IF NOT bRun THEN
	iSecondDoseCount				:= 0;
	bCycleDone 					:= FALSE;
	bCycleNotDone 				:= FALSE;	
END_IF
	
// ZASYWANIE PRZY ZJEZDZIE W DÓŁ
IF NOT bSucking AND bDoSmallSucking THEN
	mcDispencerMoveAbsolute1.Execute:= bDosingValveClosedSensor; 
	mcDispencerMoveAbsolute1.Velocity:= lrSuckVelocity;
	mcDispencerMoveAbsolute1.Position:= lrDoseVolume + 3;
	mcDispencerMoveAbsolute1.Acceleration:= lrSuckAcceleration;
	mcDispencerMoveAbsolute1.Deceleration:= lrSuckDeceleration;
	IF mcDispencerMoveAbsolute1.Done THEN
		bDoSmallSucking						:=	FALSE;
		bDoSmallSuckingDone					:=	TRUE;	
		mcDispencerMoveAbsolute1.Execute	:=	FALSE;
	END_IF
END_IF
IF  bSucking AND tonSuckValveCloseTimeDelay.Q  THEN  // [4] Opóżnienie zamknięcia zaworu ssącego [ms]                            
		bSucking := FALSE;
		mcDispencerMoveAbsolute1.Execute:= FALSE;
		bSuckingValveActuator:=FALSE;
END_IF	

ManualMovementsCleaning();
ManualMovementsPulling();
ManualMovementSync();

//ZABEZPIECZENIE PRZED UDERZENIEM W TACKĘ OCIEKOWĄ
IF DispencerLifterAxisRef.NcToPlc.ActPos	<	(lrDropCatcherHeightCV+lrDropCatcherOpenDistance-5) AND NOT bDropCatcherBackSensor THEN
	mcLifterManualMove.JogBackwards:=FALSE;
END_IF

IF (DispencerLifterAxisRef.NcToPlc.ActPos  <= 	lrDropCatcherHeightCV+(lrDropCatcherOpenDistance-5))  THEN 
	bDropCatcherActuator:=FALSE;
END_IF
END_ACTION

ACTION ManualMovementsCleaning:

(*****************CYKL MYCIA DOZOWNIKA*******************
eCleaningPreparing:=18,	//Mycie | przejazd do pozycji górnej
eCleaningReady:=19,		//Mycie | pozycja tłoka w górze
eCleaning:=20,			//Mycie | w trakcie ruchu w dół
eCleaningDone:=21		//Mycie | pozycja tłoka w dole
*********************************************************)

// Włączenie mycia
IF bManualCleaningMode  AND  (	NOT (eRunningState	=	E_DispencerState.eCleaningPreparing)		AND
								NOT (eRunningState	=	E_DispencerState.eCleaningReady) 			AND
								NOT (eRunningState	=	E_DispencerState.eCleaning)					AND
								NOT (eRunningState	=	E_DispencerState.eCleaningDone) )			THEN 
	eRunningState	:=	E_DispencerState.eCleaningPreparing;	
END_IF

//Wyłączenie mycia, zatrzymywanie
IF NOT bManualCleaningMode AND  (	eRunningState	=	E_DispencerState.eCleaningReady OR
									eRunningState	=	E_DispencerState.eCleaning OR
									eRunningState	=	E_DispencerState.eCleaningDone )	THEN

	mcDispencerStop.Execute					:= TRUE;
	bSuckingValveActuator					:= FALSE;	
	bDosingValveActuator					:= FALSE;	
	IF 	mcDispencerStop.Done THEN			
		mcDispencerStop.Execute				:= FALSE;
		eState								:= E_Station.eManualMovement;
		eRunningState						:= E_DispencerState.eReady;
	END_IF	
END_IF


//Przygotowanie
IF eRunningState=E_DispencerState.eCleaningPreparing THEN
	bSuckingValveActuator					:= TRUE;
	bDosingValveActuator					:= FALSE;
	mcDispencerMoveAbsolute1.Velocity		:= (lrDosePhase2Velocity*2)		*1.8; 	//Prędkość brana z receptury zwiększona o 30% i 2x większa niż dozowania
	mcDispencerMoveAbsolute1.Acceleration	:= lrDosePhase2Acceleration		*1.8;
	mcDispencerMoveAbsolute1.Deceleration	:= lrDosePhase2Acceleration		*1.8;
	mcDispencerMoveAbsolute1.Position		:= lrRatedDose;
	mcDispencerMoveAbsolute1.Execute		:= bSuckingValveActuator AND bSuckingValveOpenedSensor AND bDosingValveClosedSensor ;
	IF mcDispencerMoveAbsolute1.Done THEN
		mcDispencerMoveAbsolute1.Execute	:= FALSE;
		eRunningState								:= E_DispencerState.eCleaningReady;
	END_IF
END_IF


//Gotowość do mycia
IF eRunningState=E_DispencerState.eCleaningReady THEN
	bSuckingValveActuator					:= FALSE;
	bDosingValveActuator					:= FALSE;
	IF bManualCleaning THEN
		eRunningState								:= E_DispencerState.eCleaning;
	END_IF
END_IF


//Mycie, ruch w dół
IF eRunningState=E_DispencerState.eCleaning THEN
	bSuckingValveActuator					:= FALSE;
	bDosingValveActuator					:= TRUE;
	mcDispencerMoveAbsolute2.Velocity		:= lrDosePhase2Velocity			*1.8;
	mcDispencerMoveAbsolute2.Acceleration	:= lrDosePhase2Acceleration		*1.8;
	mcDispencerMoveAbsolute2.Deceleration	:= lrDosePhase2Acceleration		*1.8;
	mcDispencerMoveAbsolute2.Position		:= 0;
	mcDispencerMoveAbsolute2.Execute		:= bDosingValveActuator AND bSuckingValveClosedSensor AND bDosingValveOpenedSensor;
	IF mcDispencerMoveAbsolute2.Done THEN
		mcDispencerMoveAbsolute2.Execute	:= FALSE;
		eRunningState								:= E_DispencerState.eCleaningDone;
	END_IF	
END_IF


//Koniec mycia
IF eRunningState=E_DispencerState.eCleaningDone THEN
	bSuckingValveActuator					:= FALSE;
	bDosingValveActuator					:= FALSE;
	IF NOT bManualCleaning THEN
		eRunningState								:= E_DispencerState.eCleaningPreparing;
	END_IF
END_IF
END_ACTION

ACTION ManualMovementsPulling:
//CYKL PRZECIĄGANIA MASY
IF eRunningState=E_DispencerState.ePulling THEN
	
	IF NOT bManualPullingFast AND NOT bManualPullingSlow AND NOT bSuckingValveActuator AND NOT bDosingValveActuator AND bSuckingValveClosedSensor AND bDosingValveClosedSensor AND mcDispencerStop.Done THEN
		mcDispencerStop.Execute:=FALSE;
		mcDispencerMoveAbsolute1.Execute:=FALSE;
		mcDispencerMoveAbsolute2.Execute:=FALSE;
		bSuckingValveActuator:=FALSE;
		bDosingValveActuator:=FALSE;
		bManualPullingLatch:=FALSE;
		mcLifterManualMove.JogForward:=FALSE;
		mcLifterManualMove.JogBackwards:= FALSE;
		eState:=E_Station.eManualMovement;
		eRunningState:=E_DispencerState.eReady;
	END_IF

	mcDispencerMoveAbsolute1.Execute:=bSuckingValveActuator AND bSuckingValveOpenedSensor AND bDosingValveClosedSensor AND (bManualPullingFast OR bManualPullingSlow);
	IF mcDispencerMoveAbsolute1.Execute THEN
		;
	END_IF
	mcDispencerMoveAbsolute2.Execute:=bDosingValveActuator AND bSuckingValveClosedSensor AND bDosingValveOpenedSensor AND (bManualPullingFast OR bManualPullingSlow);
	IF bManualPullingFast THEN
		lrPullingVelocity:=300;
	ELSIF bManualPullingSlow THEN
		lrPullingVelocity:=100;
	END_IF
	mcDispencerMoveAbsolute1.Velocity:=lrPullingVelocity;
	mcDispencerMoveAbsolute2.Velocity:=lrPullingVelocity;
	
	mcDispencerMoveAbsolute1.Acceleration:=800;
	mcDispencerMoveAbsolute2.Acceleration:=800;
	mcDispencerMoveAbsolute1.Deceleration:=800;
	mcDispencerMoveAbsolute2.Deceleration:=800;
	mcDispencerMoveAbsolute1.Position:=lrRatedDose;
	mcDispencerMoveAbsolute2.Position:=0;
	
	bSuckingValveActuator:= NOT mcDispencerMoveAbsolute1.DONE AND NOT bDosingValveActuator AND  (bManualPullingFast OR bManualPullingSlow);
	bDosingValveActuator:= NOT mcDispencerMoveAbsolute2.DONE AND NOT bSuckingValveActuator AND (bManualPullingFast OR bManualPullingSlow OR mcDispencerMoveAbsolute2.Busy);
	mcDispencerStop.Execute:=NOT bSuckingValveActuator AND NOT bDosingValveActuator AND NOT bManualPullingFast AND NOT bManualPullingSlow AND eRunningState=E_DispencerState.ePulling;
END_IF
END_ACTION

ACTION ManualMovementsStepMode:
bManualLifterUp;
bManualLifterDown;
bStepMode;		
lrSetPosStepMode;

// Limity
IF lrSetPosStepMode < 1			THEN	lrSetPosStepMode := 1;	END_IF
IF lrSetPosStepMode > 10		THEN	lrSetPosStepMode := 10;	END_IF

// Zabezpieczenie przed zbyt szybkim włączaniem
tofStepModeMoving				(IN := bStepModeMoving,					PT:=T#500MS);

// Możliwe włączenie jeżeli zakończyło poprzedni ruch
rtStepModeUp					(CLK :=	bStepMode AND NOT tofStepModeMoving.Q	AND bManualLifterUp,	Q=>);
rtStepModeDown					(CLK :=	bStepMode AND NOT tofStepModeMoving.Q 	AND bManualLifterDown,	Q=>);

// Włączenie ruchu w górę
IF rtStepModeUp.Q THEN
	bStepModeMoving				:= TRUE;
	lrStepModeHeightMotorSV		:= lrLifterActualPosition	+	lrSetPosStepMode;
END_IF

// Włączenie ruchu w dół
IF rtStepModeDown.Q THEN
	bStepModeMoving				:= TRUE;
	lrStepModeHeightMotorSV		:= lrLifterActualPosition	-	lrSetPosStepMode;
END_IF
// DODAĆ RESET bStepModeMoving PO BLEDZIE!
// Ruch w górę !SPRAWDZIC ZNAKI!
IF bStepModeMoving THEN
	mcLifterManualMove.JogForward		:=	lrLifterActualPosition	<=	lrStepModeHeightMotorSV;
	mcLifterManualMove.JogBackwards		:=	lrLifterActualPosition	>=	lrStepModeHeightMotorSV;	
	
	IF ABS(lrLifterActualPosition-lrStepModeHeightMotorSV) < 0.5	OR	// Pozycja osiągnięta (co do 1mm)
			(lrLifterActualPosition<=lrMinPosition)					OR 	// Pozycja poniżej minimalnej
			(lrLifterActualPosition>=lrMaxPosition) 					// Pozycja powyżej maksymalnej
	THEN
		mcLifterManualMove.JogForward	:= FALSE;
		mcLifterManualMove.JogForward	:= FALSE;
		bStepModeMoving					:= FALSE;
		bManualLifterUp					:= FALSE;
		bManualLifterDown				:= FALSE;
	END_IF	
END_IF
END_ACTION

ACTION ManualMovementSync:
//Przygotowanie
IF bManualSync THEN
	
CASE iManualSyncCase OF
	
	0:	
		//Rozpoczęcie
		IF bManualSync THEN
			iManualSyncCase	:=	iManualSyncCase	+	10;
		END_IF

	10:
		
			//Ruch tłokiem
			IF ABS(DispencerAxisRef.NcToPlc.ActPos-lrDoseVolume)>1 THEN //Nie wykonuj nie potrzebnie ruchu jeżeli już jest na pozycji
				bSuckingValveActuator				:= ABS(DispencerAxisRef.NcToPlc.ActPos-lrDoseVolume)>1;
			END_IF
			bDosingValveActuator					:= FALSE;
			mcDispencerMoveAbsolute1.Velocity		:= (lrDosePhase2Velocity*2)		*1.8; 	//Prędkość brana z receptury zwiększona o 30% i 2x większa niż dozowania
			mcDispencerMoveAbsolute1.Acceleration	:= lrDosePhase2Acceleration		*1.8;
			mcDispencerMoveAbsolute1.Deceleration	:= lrDosePhase2Acceleration		*1.8;
			mcDispencerMoveAbsolute1.Position		:= lrDoseVolume;
			mcDispencerMoveAbsolute1.Execute		:= bSuckingValveActuator AND bSuckingValveOpenedSensor AND bDosingValveClosedSensor ;

		//Ruch podnośnikiem
		IF bDispencerWithLifter THEN
			IF NOT bLifterIsNearReadyPosition THEN
				bDropCatcherActuator 				:= FALSE;			
				IF bDropCatcherBackSensor THEN
					mcLifterMoveAbsolute.Execute	:= TRUE;
				END_IF		
				mcLifterMoveAbsolute.Acceleration	:= lrLifterAcceleration/15;
				mcLifterMoveAbsolute.Velocity		:= lrLifterVelocity/15;
				mcLifterMoveAbsolute.Position		:= lrLifterReadyPosition;
			END_IF	
		END_IF
		
		//Wykonano ruchhy
		IF 
			(mcDispencerMoveAbsolute1.Done OR ABS(DispencerAxisRef.NcToPlc.ActPos-lrDoseVolume)<=1) AND	//Wykonano ruch tłokiem 
			(NOT bDispencerWithLifter OR mcLifterMoveAbsolute.Done OR bLifterIsNearReadyPosition)		//Wykonano ruhc podnośnikiem
		THEN
			mcDispencerMoveAbsolute1.Execute	:=	FALSE;
			mcLifterMoveAbsolute.Execute		:=	FALSE;
			iManualSyncCase						:=	iManualSyncCase	+	10;
		END_IF	
		
	20:
		//Koniec
		bManualSync								:=	FALSE;
		iManualSyncCase							:=	0;
	
	
END_CASE



END_IF
END_ACTION

ACTION ResetCommands:
bStepModeMoving		:=	FALSE;



//Synchornizacja
iManualSyncCase		:= 0;
bManualSync			:= FALSE;


iSecondDoseCount	:=	0;

//GoingUp
iCaseGoingUp					:=	0;
mcLifterMoveAbsolute2.Execute	:=	FALSE;


// Pogrzybie
mcDispencerSoftReset.Execute	:= FALSE;
END_ACTION

ACTION Running:
//	100					300			250
IF lrDosePhase1Volume>lrDoseVolume-lrDosePhase2Volume THEN
	lrDosePhase1Volume:=lrDoseVolume-lrDosePhase2Volume;
END_IF
// 200					300			200
IF lrDosePhase2Volume>lrDoseVolume-lrDosePhase1Volume THEN
	lrDosePhase2Volume:=lrDoseVolume-lrDosePhase1Volume;
END_IF

tonbDispenserSim(in:=(bSimDoser AND eRunningState = 6 AND bDispencerWithLifter AND ((mcLifterMoveAbsolute.Done OR NOT bDispencerWithLifter)  
					AND (mcDispencerMoveAbsolute1.Done OR ABS(LREAL_TO_DINT(DispencerAxisRef.NcToPlc.ActPos)-LREAL_TO_DINT(lrDoseVolume))<=1 OR bDoSmallSuckingDone)) 
					AND bMultiMasterSyncIn) , PT:=T#300MS);
tonbDispencerLifterSim (in:=bDispencerWithLifter AND bSimDoser AND eRunningState = 6,PT:=T#300MS); 
(*Ograniczenia GearRatio*)
IF eRunningState = E_DispencerState.eReady THEN
	lrGearRatio:=-ABS(lrLifterStopDosePosition-lrLifterStartDosePosition+0.000000000001)
								/(*---------------------------------------------------------------------*)
								((BOOL_TO_INT(bLiftSynchroPh1)*lrDosePhase1Volume)
								+(BOOL_TO_INT(bLiftSynchroPh2)*(lrDoseVolume-lrDosePhase2Volume-lrDosePhase1Volume))
								+((BOOL_TO_INT(bLiftSynchroPh3)*lrDosePhase2Volume))
								+ 0.000000000001); 
	IF bLiftSynchroPh3 AND lrGearRatio<-1.2 THEN
		lrGearRatio:=-1.2;
	END_IF
END_IF
(*Koniec Ograniczenia GearRatio*)

							

CASE eRunningState OF

//====================================
	
	(*Oczekiwanie na wykonanie pojedynczego cyklu*)
	E_DispencerState.eReady:
                                         	
		IF NOT bCycleDone AND NOT bCycleNotDone THEN                                           	
			IF bRun THEN                				
				eRunningState		:=	E_DispencerState.ePreparingToDose;
				lrSuckingMassStart	:=	DispencerAxisRef.NcToPlc.ActPos;
				iCaseGoingUp		:=	0;
			END_IF
		END_IF
		
		bMultiMasterSyncOut:=FALSE;
		
//====================================		
				
	E_DispencerState.ePreparingToDose:

				//Jeśli oś w stanie 'master' przy gearing przejdź do stanu fazy pierwszej dozowania
				IF bDispencerWithLifter AND (NOT bSimDoser OR tonbDispencerLifterSim.Q)THEN
					bDropCatcherActuator:=FALSE;
					mcLifterStop.Execute:=FALSE;
					mcLifterMoveAbsolute.Execute:= NOT mcLifterStop.Done AND bDropCatcherBackSensor AND bDropCatcherActuator=FALSE;
					mcLifterMoveAbsolute.Deceleration	:=	lrLifterDeceleration;
					mcLifterMoveAbsolute.Acceleration	:=	lrLifterAcceleration;
					mcLifterMoveAbsolute.Velocity		:=	lrLifterVelocity;
					mcLifterMoveAbsolute.Position		:=	lrLifterStartDosePosition;
				END_IF
				
				mcDispencerStop.Execute:=FALSE;
				//IF ABS(LREAL_TO_DINT(DispencerAxisRef.NcToPlc.ActPos)-LREAL_TO_DINT(lrDoseVolume))>1 THEN //Zmiana dp
				IF NOT bDoSmallSuckingDone THEN
					mcDispencerMoveAbsolute1.Execute:= NOT mcDispencerStop.BUSY;
					mcDispencerMoveAbsolute1.Velocity:= lrSuckVelocity;
					mcDispencerMoveAbsolute1.Position:= lrDoseVolume;
					mcDispencerMoveAbsolute1.Acceleration:= lrSuckAcceleration;
					mcDispencerMoveAbsolute1.Deceleration:= lrSuckDeceleration;
					//END_IF;	
				END_IF
				
				bMultiMasterSyncOut:=(mcDispencerMoveAbsolute1.Done OR bDoSmallSuckingDone) 
				AND ((ABS(DispencerLifterAxisRef.NcToPlc.ActPos)-lrLifterStartDosePosition)<=1);

					//Jeśli osiągnięta pozycja zassania i jeśli jest podnośnik dozownika
//dp				IF (mcLifterMoveAbsolute.Done OR NOT bDispencerWithLifter)  AND (mcDispencerMoveAbsolute1.Done OR ABS(LREAL_TO_DINT(DispencerAxisRef.NcToPlc.ActPos)-LREAL_TO_DINT(lrDoseVolume))<=1(*(LREAL_TO_DINT(DispencerAxisRef.NcToPlc.ActPos)=LREAL_TO_DINT(lrDoseVolume))*)) 
					IF ((mcLifterMoveAbsolute.Done OR NOT bDispencerWithLifter)  
					AND (mcDispencerMoveAbsolute1.Done OR ABS(LREAL_TO_DINT(DispencerAxisRef.NcToPlc.ActPos)-LREAL_TO_DINT(lrDoseVolume))<=1 OR bDoSmallSuckingDone)) 

					AND bMultiMasterSyncIn
					//AND (NOT bSimDoser OR tonbDispenserSim.Q)
						THEN
			    	
					//Jeśli nalewarka ma podnośnik i wybrana któraś z opcji ruchu synchronicznego przejdź do procedury zasprzęglania
						IF bDispencerWithLifter AND (bLiftSynchroPh1 OR bLiftSynchroPh2 OR bLiftSynchroPh3) THEN
							mcLifterGearIn.Acceleration:=lrLifterAcceleration;
							mcLifterGearIn.Deceleration:=lrLifterDeceleration;
							mcLifterGearIn.Jerk:=lrLifterDeceleration;
							mcLifterGearIn.GearRatio:=0.0000000001;
						END_IF
						bSucking:=FALSE; //ZASYSANIE PODCZAS ZJAZDU
						bSuckingValveActuator:=FALSE; //ZASYSANIE PODCZAS ZJAZDU
						eRunningState:=E_DispencerState.eDosingPh1;
						mcLifterMoveAbsolute.Execute:=FALSE;
						mcDispencerMoveAbsolute1.Execute:= FALSE;
						mcDispencerMoveAbsolute2.Execute:= FALSE;
						mcDispencerMoveAbsolute3.Execute:= FALSE;
						lrStartDosingPos:=DispencerAxisRef.NcToPlc.ActPos;
						bDoSmallSuckingDone := FALSE;
					END_IF

//====================================					
	
	E_DispencerState.eDosingPh1:
				bDropCatcherActuator:=FALSE;
	
				IF bDispencerWithLifter AND (bLiftSynchroPh1 OR bLiftSynchroPh2 OR bLiftSynchroPh3) AND NOT mcLifterGearIn.Enable THEN
					mcLifterGearIn.Enable:= NOT mcDispencerMoveAbsolute1.Busy;
				END_IF
				
				IF (mcLifterGearIn.InGear OR NOT bDispencerWithLifter OR NOT( bLiftSynchroPh1 OR bLiftSynchroPh2 OR bLiftSynchroPh3 )) THEN
					mcDispencerMoveAbsolute1.Execute:= bDropCatcherBackSensor AND tonDoseValveOpenTimeAcc.Q;
					mcDispencerMoveAbsolute1.Velocity:= lrDosePhase1Velocity;
					mcDispencerMoveAbsolute1.Position:= lrDoseVolume-lrDosePhase1Volume;
					mcDispencerMoveAbsolute1.Acceleration:= lrDosePhase1Acceleration;
					mcDispencerMoveAbsolute1.Deceleration:= lrDosePhase1Deceleration;
					mcDispencerMoveAbsolute1.BufferMode:= MC_BlendingPrevious;
				END_IF;	
				
				IF bDispencerWithLifter THEN
					IF NOT bLiftSynchroPh1 THEN
						mcLifterGearIn.GearRatio:=0.00000000001;
					ELSE
						mcLifterGearIn.GearRatio:=lrGearRatio;
					END_IF
				END_IF
				//Jeśli zakręcarka na wysokości zakręcania przejdź do stanu zakręcania
				IF (mcLifterGearIn.InGear OR NOT bDispencerWithLifter OR NOT( bLiftSynchroPh1 OR bLiftSynchroPh2 OR bLiftSynchroPh3 )) 
				AND mcDispencerMoveAbsolute1.Execute AND (mcDispencerMoveAbsolute1.Busy OR mcDispencerMoveAbsolute1.Done)
				(*AND lrDosePhase2Volume>lrDosePhase2Volume*) THEN
					
					mcDispencerMoveAbsolute2.Execute:= bDropCatcherBackSensor;
					mcDispencerMoveAbsolute2.Velocity:= lrDosePhase2Velocity;
					mcDispencerMoveAbsolute2.Position:= lrDosePhase2Volume;
					mcDispencerMoveAbsolute2.Acceleration:= lrDosePhase2Acceleration;
					mcDispencerMoveAbsolute2.Deceleration:= lrDosePhase2Deceleration;
					mcDispencerMoveAbsolute2.BufferMode:= MC_BlendingPrevious;
				END_IF
				
				IF mcDispencerMoveAbsolute1.Done AND mcDispencerMoveAbsolute1.Execute THEN
					//mcDispencerMoveAbsolute1.Execute:= FALSE;
					eRunningState:=E_DispencerState.eDosingPh2;
				END_IF
			
	//====================================					
	
	E_DispencerState.eDosingPh2:
	
				IF (mcLifterGearIn.InGear OR NOT bDispencerWithLifter OR NOT( bLiftSynchroPh1 OR bLiftSynchroPh2 OR bLiftSynchroPh3 )) 
					AND mcDispencerMoveAbsolute2.Execute AND (mcDispencerMoveAbsolute2.Busy OR mcDispencerMoveAbsolute2.Done)
							(*AND lrDoseVolume>lrDosePhase2Volume*) THEN	
(*					mcDispencerMoveAbsolute1.Execute:= bDropCatcherBackSensor;
					mcDispencerMoveAbsolute1.Velocity:= lrDosePhase3Velocity;
					mcDispencerMoveAbsolute1.Position:= 0;
					mcDispencerMoveAbsolute1.Acceleration:= lrDosePhase3Acceleration;
					mcDispencerMoveAbsolute1.Deceleration:= lrDosePhase3Deceleration;
					mcDispencerMoveAbsolute1.BufferMode:= MC_BlendingNext;*)
					mcDispencerMoveAbsolute3.Execute:= bDropCatcherBackSensor;
					mcDispencerMoveAbsolute3.Velocity:= lrDosePhase3Velocity;
					mcDispencerMoveAbsolute3.Position:= 0;
					mcDispencerMoveAbsolute3.Acceleration:= lrDosePhase3Acceleration;
					mcDispencerMoveAbsolute3.Deceleration:= lrDosePhase3Deceleration;
					mcDispencerMoveAbsolute3.BufferMode:= MC_BlendingPrevious;
				END_IF
				
				IF bDispencerWithLifter THEN
					IF NOT bLiftSynchroPh2 THEN
						mcLifterGearIn.GearRatio:=0.00000000001;
					ELSE
						mcLifterGearIn.GearRatio:=lrGearRatio;
					END_IF
				END_IF
				
				//IF mcDispencerMoveAbsolute2.Done AND bTest THEN
				IF mcDispencerMoveAbsolute2.Done AND mcDispencerMoveAbsolute2.Execute  THEN					
					//mcDispencerMoveAbsolute2.Execute:= FALSE;
					IF bDoSecondDose AND iSecondDoseCount >=1 THEN
						bDoSecondDose	:=	FALSE;
					END_IF	
			
					iSecondDoseCount	:=	iSecondDoseCount	+	1;
					eRunningState		:=	E_DispencerState.eDosingPh3;

				END_IF
					
	//====================================	
				
	//FAZA TRZECIA DOZOWANIA
	E_DispencerState.eDosingPh3:
														
		IF bDispencerWithLifter THEN
			IF NOT bLiftSynchroPh3 THEN
				mcLifterGearIn.GearRatio:=0.00000000001;
			ELSE
				mcLifterGearIn.GearRatio:=lrGearRatio;
			END_IF
		END_IF
		(*n*)
		bMultiMasterSyncOut:=NOT mcDispencerMoveAbsolute3.Done;
		
		IF mcDispencerMoveAbsolute3.Done AND (tonDoseValveCloseTimeDec.Q OR bDoseSucking) AND (NOT bMultiMasterSyncIn OR bSimDoser) THEN
			
			nCountTest12:=nCountTest12+1;
			lrSuckingMassStart:=DispencerAxisRef.NcToPlc.ActPos;
			mcDispencerMoveAbsolute1.Execute:= FALSE;
			mcDispencerMoveAbsolute2.Execute:= FALSE;
			mcDispencerMoveAbsolute3.Execute:= FALSE;
			IF bDispencerWithLifter THEN (*n*)
				mcLifterGearOut.Execute:=TRUE;
				mcLifterGearIn.Enable:=FALSE;
			END_IF
			
			IF bDoseSucking THEN (*n*)
				eRunningState	:=	E_DispencerState.eDoseSucking;
			ELSE
				iCaseGoingUp	:=	0;
				eRunningState	:=	E_DispencerState.eGoingUp; 
			END_IF
			
			IF	bDoSecondDose THEN
				eRunningState	:=	E_DispencerState.eSucking; 				
			END_IF
			
			bDosingValveActuator:=FALSE;
		END_IF
		
	//====================================	
			
	E_DispencerState.eDoseSucking:
					mcDispencerMoveAbsolute1.Execute:= bDosingValveOpenedSensor AND tonDoseSuckingTimeDelay.Q; // [6] [Podsysanie] Opóźnienie podsysania [ms]
					mcDispencerMoveAbsolute1.Velocity:= lrLifterVelocity;
					mcDispencerMoveAbsolute1.Position:= lrDoseSuckingVolume;
					mcDispencerMoveAbsolute1.Acceleration:= lrLifterAcceleration;
					mcDispencerMoveAbsolute1.Deceleration:= lrLifterDeceleration;
					IF  mcDispencerMoveAbsolute1.Done THEN
						mcDispencerMoveAbsolute2.Execute:= FALSE;
						mcDispencerMoveAbsolute3.Execute:= FALSE;
					END_IF				
					//Zmiana na mcLifterMoveAbsolute2, bylo 1
					IF bDispencerWithLifter AND tonDoseValveCloseTimeDec.Q THEN	// [2] Opóźnienie zamknięcia zaworu tłoczenia [ms]

						mcLifterMoveAbsolute2.Execute:= TRUE; 
						mcLifterMoveAbsolute2.Velocity:= lrLifterVelocity;
						mcLifterMoveAbsolute2.Position:= lrLifterReadyPosition;
						mcLifterMoveAbsolute2.Acceleration:= lrLifterAcceleration;
						mcLifterMoveAbsolute2.Deceleration:= lrLifterDeceleration;

						IF nDosingDoneDelayTime > 0 THEN //Nowe
							mcLifterMoveAbsolute2.Position		:=	lrCatchHeightSV + 5;
						ELSE
							mcLifterMoveAbsolute2.Position		:= lrLifterReadyPosition;
						END_IF						
												
						
					END_IF
					//DP CZY TUTAJ DODAĆ LIFTER DONE?
					IF mcDispencerMoveAbsolute1.Done AND tonDoseValveCloseTimeDec.Q THEN // [2] Opóźnienie zamknięcia zaworu tłoczenia [ms]		
						eRunningState:=E_DispencerState.eDoseSuckingDone;
						mcDispencerMoveAbsolute1.Execute:= FALSE;
					END_IF		
	

	//====================================

	E_DispencerState.eDoseSuckingDone:
	
				iCaseGoingUp	:=	0;
				eRunningState	:=	E_DispencerState.eGoingUp;
						
		
//====================================					
	
	//DOZOWANIE WYKONANE
	//Zaczyna sie zasysanie i podnoszenie jesli bDispencerWithLifter. Po zaniku bDose, przechodzi do nastepnych stanów	
	E_DispencerState.eGoingUp:
				IF mcLifterGearOut.Done THEN //DP NOWE
					mcLifterGearOut.Execute:=FALSE;
				END_IF
	
				btestgoingup:=btestgoingup+1;
				IF bDispencerWithLifter AND NOT mcLifterGearOut.Done THEN
					IF NOT mcLifterGearInEnable AND NOT mcDispencerMoveAbsolute1.Execute THEN
						mcDispencerMoveAbsolute1.Execute:= bDosingValveClosedSensor AND tonSuckValveOpenTimeDelay.Q; // [3] Opóżnienie rozpoczęcia ssania po tłoczeniu [ms]
						mcDispencerMoveAbsolute1.Velocity:= lrSuckVelocity;
						mcDispencerMoveAbsolute1.Position:= lrDoseVolume;
						mcDispencerMoveAbsolute1.Acceleration:= lrSuckAcceleration;
						mcDispencerMoveAbsolute1.Deceleration:= lrSuckDeceleration;
					END_IF
					
					
					CASE iCaseGoingUp OF
						
						0:
							iCaseGoingUp	:=	iCaseGoingUp	+	10;
						
						10:
							IF NOT mcLifterGearOut.Execute THEN
								//IF nDosingDoneDelayTime > 0  THEN
								IF nDosingDoneDelayTime > 0 AND NOT bDoseSucking THEN	//Nowe								
									mcLifterMoveAbsolute2.Execute		:=	TRUE;
									mcLifterMoveAbsolute2.Acceleration	:=	lrLifterAcceleration;
									mcLifterMoveAbsolute2.Deceleration	:=	lrLifterDeceleration;					
									mcLifterMoveAbsolute2.Velocity		:=	lrLifterVelocity;
//									mcLifterMoveAbsolute2.Position		:=	lrCatchHeightSV - 5;
									mcLifterMoveAbsolute2.Position		:=	lrCatchHeightSV + 20;									
									mcLifterMoveAbsolute2.BufferMode	:=	MC_BlendingPrevious;
									iCaseGoingUp						:=	iCaseGoingUp	+	10;
								ELSE
									iCaseGoingUp	:=	100;
								END_IF
							END_IF
						20:
							IF mcLifterMoveAbsolute2.Done THEN
								iCaseGoingUp						:=	iCaseGoingUp	+	10;
							END_IF

						30:
							IF tonDosingDoneDelay.Q THEN
								iCaseGoingUp	:=	100;
							END_IF					
						100:
							mcLifterMoveAbsolute.Execute		:=	TRUE;
							//mcLifterMoveAbsolute.Execute:= tonDosingDoneDelay.Q;//
							mcLifterMoveAbsolute.Acceleration	:=	lrLifterAcceleration/4;// /2
							mcLifterMoveAbsolute.Deceleration	:=	lrLifterDeceleration;	// /2				
							mcLifterMoveAbsolute.Velocity		:=	lrLifterVelocity/2; // /2
							mcLifterMoveAbsolute.Position		:=	lrLifterReadyPosition;
							mcLifterMoveAbsolute.BufferMode		:=	MC_BlendingPrevious;
							//Koniec ruchu
						
					END_CASE	
					
				ELSE
					mcDispencerMoveAbsolute1.Execute:= bDosingValveClosedSensor;
					mcDispencerMoveAbsolute1.Velocity:= lrSuckVelocity;
					mcDispencerMoveAbsolute1.Position:= lrDoseVolume;
					mcDispencerMoveAbsolute1.Acceleration:= lrSuckAcceleration;
					mcDispencerMoveAbsolute1.Deceleration:= lrSuckDeceleration;
				END_IF
				// [3] Opóżnienie rozpoczęcia ssania po tłoczeniu [ms]
				IF	tonSuckValveOpenTimeDelay.Q AND (mcLifterMoveAbsolute.Done OR NOT bDispencerWithLifter) AND (lrLifterActualPosition>lrLifterReadyPosition-5 AND lrLifterActualPosition<lrLifterReadyPosition+5) AND 
					(iCaseGoingUp	>=	100 OR NOT bDispencerWithLifter)
				THEN
					iCaseGoingUp	:=	0;
					mcLifterMoveAbsolute2.Execute:=	FALSE;
					mcLifterMoveAbsolute.Execute:= FALSE;
					eRunningState:=E_DispencerState.eDosingDone;	
				END_IF
  	
//====================================				
		
	E_DispencerState.eDosingDone:
	
		bDoSmallSucking :=	bDoSmallSuckingOption; //Test dodatkowego zasysania
	
		mcDispencerMoveAbsolute1.Execute:= bDosingValveClosedSensor;
		mcDispencerMoveAbsolute1.Velocity:= lrSuckVelocity;
		mcDispencerMoveAbsolute1.Position:= lrDoseVolume;
		mcDispencerMoveAbsolute1.Acceleration:= lrSuckAcceleration;
		mcDispencerMoveAbsolute1.Deceleration:= lrSuckDeceleration;
		mcDispencerMoveAbsolute1.BufferMode:= MC_Buffered; //ZMIANA BUFFERMODE
			
		IF mcDispencerMoveAbsolute1.Done AND tonSuckValveCloseTimeDelay.Q (*AND tonDosingDoneDelay.Q*) THEN // [4] Opóżnienie zamknięcia zaworu ssącego [ms]
			bSuckingValveActuator:=FALSE;
			mcDispencerMoveAbsolute1.Execute:=FALSE;
			eRunningState:=E_DispencerState.eReady;
			bCycleDone := TRUE;
		ELSE
			eRunningState:=E_DispencerState.eSucking;	
		END_IF	

//====================================		
	
	E_DispencerState.eSucking:
			mcDispencerMoveAbsolute1.Execute:= bDosingValveClosedSensor; 
			mcDispencerMoveAbsolute1.Velocity:= lrSuckVelocity;
			mcDispencerMoveAbsolute1.Position:= lrDoseVolume;
			mcDispencerMoveAbsolute1.Acceleration:= lrSuckAcceleration;
			mcDispencerMoveAbsolute1.Deceleration:= lrSuckDeceleration;
			bSucking := TRUE;	
			// ZASYWANIE PRZY ZJEZDZIE W DÓŁ
			//IF  (*mcDispencerMoveAbsolute1.Done AND  tonSuckValveCloseTimeDelay.Q AND*) tonDosingDoneDelay.Q THEN  // [4] Opóżnienie zamknięcia zaworu ssącego [ms]                            
					//mcDispencerMoveAbsolute1.Execute:= FALSE;
					mcDispencerMoveAbsolute2.Execute:= FALSE;
					mcDispencerMoveAbsolute3.Execute:= FALSE;
					//bSuckingValveActuator:=FALSE;
					IF bDoSecondDose THEN
						eRunningState	:=	E_DispencerState.ePreparingToDose;	
					ELSE
						eRunningState	:=	E_DispencerState.eReady;	
						bCycleDone		:=	TRUE;
					END_IF
			//END_IF		

END_CASE
		



		//Tłoczący
		IF eRunningState=E_DispencerState.eDosingPh1 OR eRunningState=E_DispencerState.eDosingPh2 OR eRunningState=E_DispencerState.eDosingPh3 OR 
		   eRunningState=E_DispencerState.eDoseSucking THEN
			
			bDosingValveActuator:= (lrStartDosingPos-lrDosingValveOpenVolume>=LREAL_TO_INT(DispencerAxisRef.NcToPlc.ActPos))AND(lrDosingValveCloseVolume<=LREAL_TO_INT(DispencerAxisRef.NcToPlc.ActPos));
			bSuckingValveActuator:=FALSE;
			
			IF (lrDosingValveOpenVolume+lrDosingValveCloseVolume)>(lrStartDosingPos)  THEN
				bDosingValveActuator:=TRUE;	
				nCheckCount125:=nCheckCount125+1;
			END_IF
			
			IF  lrDoseValveOpenTimeAcc > 0 THEN // [1] Przyśpieszenie otwarcia zaworu tłoczenia [ms]
				bDosingValveActuator:=TRUE;	
				nCheckCount124:=nCheckCount124+1;
			END_IF
										//bylo = (tonDoseValveCloseTimeDec.Q OR bDoseSucking) 
			IF (lrDosingValveCloseVolume>LREAL_TO_INT(DispencerAxisRef.NcToPlc.ActPos)) AND (lrDoseValveCloseTimeDec = 0 AND NOT bDoseSucking) THEN 
				bDosingValveActuator:=FALSE;
				nCheckCount123:=nCheckCount123+1;
			END_IF
			ninttest:=LREAL_TO_INT(DispencerAxisRef.NcToPlc.ActPos);
		END_IF
		
		
		
		//Ssący																								
		IF eRunningState=E_DispencerState.ePreparingToDose OR 
			eRunningState=E_DispencerState.eSucking  OR  
			(*eState=E_DispencerState.eDosingDone OR *)
			eRunningState=E_DispencerState.eGoingUp OR
			bSucking 
 			(*OR
			eState=E_DispencerState.eDoseSuckingDone*) (*AND mcDispencerMoveAbsolute1.Busy*) 
		 THEN
			
			bSuckingValveActuator:=(((ABS(LREAL_TO_INT(lrSuckingMassStart-DispencerAxisRef.NcToPlc.ActPos)))>LREAL_TO_INT(lrSuckValveOpenVolume))
									AND((ABS(LREAL_TO_INT(lrDoseVolume-DispencerAxisRef.NcToPlc.ActPos)))>LREAL_TO_INT(lrSuckValveCloseVolume))); 
																					
			IF lrDoseValveOpenTimeAcc >= 0 THEN // [1] Przyśpieszenie otwarcia zaworu tłoczenia [ms] (Dodatkowe zabezpieczenie bo czasami sie na chwile zamykał)
				bDosingValveActuator:=FALSE;
				nCheckCount1263:=nCheckCount1236+1;
			END_IF 
			
			IF	(lrSuckValveOpenVolume+lrSuckValveCloseVolume)>(ABS(lrDoseVolume-lrSuckingMassStart)) AND (lrSuckValveOpenVolume > mcDispencerMoveAbsolute1.Position) AND 
				(lrSuckValveCloseVolume < mcDispencerMoveAbsolute1.Position)  THEN
				bSuckingValveActuator:=TRUE;	
				nCheckCount1234:=nCheckCount1234+1;
			END_IF
			// [4] Opóżnienie zamknięcia zaworu ssącego [ms]
//dp		IF NOT tonSuckValveCloseTimeDelay.Q AND (eRunningState=E_DispencerState.eDosingDone OR eRunningState=E_DispencerState.eSucking) AND lrSuckValveCloseVolume = 0 THEN (*4*)
			IF NOT tonSuckValveCloseTimeDelay.Q AND (eRunningState=E_DispencerState.eDosingDone OR eRunningState=E_DispencerState.eSucking) AND lrSuckValveCloseVolume = 0 AND (*4*)
			((ABS(LREAL_TO_INT(lrSuckingMassStart-DispencerAxisRef.NcToPlc.ActPos)))>LREAL_TO_INT(lrSuckValveOpenVolume)) THEN
				bSuckingValveActuator:=TRUE;	
				nCheckCount1233:=nCheckCount1233+1;
			END_IF
			//IF NOT tonSuckValveOpenTimeDelay.Q AND eState=E_DispencerState.eGoingUp THEN										
			IF NOT tonSuckValveOpenTimeDelay.Q AND eRunningState=E_DispencerState.eGoingUp THEN
				bSuckingValveActuator:=FALSE;	
				nCountCheckDisp1:=nCountCheckDisp1+1;
			END_IF
			
			IF (lrSuckValveCloseTimeDelay>0 AND tonSuckValveOpenTimeDelay.Q) AND eRunningState=E_DispencerState.eGoingUp THEN
				bSuckingValveActuator:=TRUE;	
				nCheckCount1235:=nCheckCount1235+1;
			END_IF
			
			IF bSucking THEN
				bSuckingValveActuator	:= TRUE;
			END_IF
			
		END_IF
END_ACTION

ACTION SecondDose:

lrLifterStartDosePosition;
lrLifterStopDosePosition;


IF lrDoseVolume	>	lrRatedDose THEN
	bSecondDoseMode		:=TRUE;

	IF iSecondDoseCount = 0 THEN
		bDoSecondDose				:=	TRUE;
		lrDoseVolume 				:=	lrDoseVolume / 2 ;
		lrLifterStartDosePosition	;
		lrLifterStopDosePosition	:=	((lrLifterStopDosePosition - lrLifterStartDosePosition) / 2 ) + lrLifterStartDosePosition;
		
	ELSIF iSecondDoseCount >=1 THEN
		lrDoseVolume 				:=	lrDoseVolume / 2 ;
		lrLifterStartDosePosition	:=	((lrLifterStopDosePosition - lrLifterStartDosePosition) / 2 ) + lrLifterStartDosePosition;
		lrLifterStopDosePosition	;
		
	END_IF
	
ELSIF eState = E_Station.eReady  OR bCycleDone THEN
	bSecondDoseMode					:=	FALSE;
	bDoSecondDose					:=	FALSE;
END_IF
END_ACTION

ACTION Signals:

bLifterIsNearReadyPosition := ABS(lrLifterActualPosition-lrLifterReadyPosition) < 2 ;
END_ACTION

ACTION Statistics:
IF LREAL_TO_INT(lrStartDosingPos)<> LREAL_TO_INT(lrLifterReadyPosition) THEN
	rtrigCycleTimerRead(CLK:=LREAL_TO_INT(lrLifterActualPosition) = LREAL_TO_INT(lrLifterReadyPosition));
	IF rtrigCycleTimerRead.Q THEN
			tCycleTime:=tonCycleTimer.ET;
	END_IF
	tonCycleTimer(IN:=LREAL_TO_INT(lrLifterActualPosition) <> LREAL_TO_INT(lrLifterReadyPosition),PT:=T#1D);
ELSE
	rtrigCycleTimerRead(CLK:=bCycleDone);
	IF rtrigCycleTimerRead.Q THEN
		tCycleTime:=tonCycleTimer.ET;
	END_IF
	tonCycleTimer(IN:=eRunningState>E_DispencerState.eReady,PT:=T#1D);
END_IF
END_ACTION

END_FUNCTION_BLOCK

// ---- POUs/FB/FB_HomingTorque.TcPOU
//==================================================================================================
//							Beckhoff Automation Poland
//									3.01.2022
//	Function block running home procedure in torque mode
//	Avaliable two modes:
//	1. Lag based - bLagBased = TRUE - define lrLagLimit which decides about end of movement
//	2. Torque based - bLagBased = FALSE - define lrTorqueLimit and lrTorqueTolerance which decides about end of movement
//
//	Library: Tc3_MC2_AdvancedHoming, Tc2_MC2, 
//
//  v1.0	|| TC v 3.1.4024.22		|| First edition 
//==================================================================================================
FUNCTION_BLOCK FB_HomingTorque
VAR_IN_OUT
	Axis 										: Tc2_MC2.AXIS_REF;
END_VAR  
VAR_INPUT
	bExecute									: BOOL;
	bLagBased									: BOOL;					// TRUE: MC_StepBlockLagBased, FALSE: MC_StepBlock
	eDirection									: Tc3_MC2_AdvancedHoming.MC_Home_Direction;
	lrVelocity									: LREAL;
	lrSetPosition								: LREAL;
	lrDetectionVelocityLimit					: LREAL;
	tDetectionVelocityTime						: TIME;
	tTimeLimit									: TIME;
	lrDistanceLimit								: LREAL;
	lrTorqueLimit								: LREAL;
	lrTorqueTolerance							: LREAL;
	lrLagLimit									: LREAL;
	lrDistance									: LREAL;
END_VAR                             		
VAR_OUTPUT                              		
	bDone										: BOOL;
	bBusy										: BOOL;
	bCommandAborted								: BOOL;
	bError										: BOOL;
	udiErrorID									: UDINT;
END_VAR
VAR
//=========================== Common ============================
	nStep										: UDINT;
	stParameter									: Tc3_MC2_AdvancedHoming.MC_HomingParameter;
	stOptions									: Tc3_MC2_AdvancedHoming.ST_Home_Options3;
//========================= Step Block ==========================
	mcStepBlock									: Tc3_MC2_AdvancedHoming.MC_StepBlock;
	mcStepBlockLag								: Tc3_MC2_AdvancedHoming.MC_StepBlockLagBased;
//=========================== Finish ============================
	mcFinishHoming								: Tc3_MC2_AdvancedHoming.MC_FinishHoming;
//============================ Abort ============================
	mcAbortHoming								: Tc3_MC2_AdvancedHoming.MC_AbortHoming;
//========================== Internal ===========================
    {attribute 'hide'}
	udiErrorID_Int								: UDINT;
//===============================================================
END_VAR

//====== Call FBs outside CASE - easier debugging ===============
mcStepBlockLag(Axis								:= Axis, 
				Parameter						:= stParameter);
				                        		
mcStepBlock(	Axis							:= Axis, 
				Parameter						:= stParameter);	
                                        		
mcFinishHoming(	Axis							:= Axis, 
				Parameter						:= stParameter);
				                        	
mcAbortHoming(	Axis							:= Axis, 
				Parameter						:= stParameter);
				
//============== CASE instruction - step machine ================
CASE nStep OF
	
	0: // Wait for command
	
		IF bExecute THEN
			bBusy								:= TRUE;
			// Latch finish parameters
			mcFinishHoming.Distance				:= lrDistance;
			mcFinishHoming.Velocity				:= lrVelocity;
				
			IF bLagBased THEN

				mcStepBlockLag(Axis				:= Axis, 
						Parameter				:= stParameter, 
						Execute					:= TRUE, 
						Direction				:= eDirection, 
						Velocity				:= lrVelocity,
						SetPosition				:= lrSetPosition, 
						DetectionVelocityLimit	:= lrDetectionVelocityLimit, 
						DetectionVelocityTime	:= tDetectionVelocityTime, 
						TimeLimit				:= tTimeLimit, 
						DistanceLimit			:= lrDistanceLimit, 
						TorqueLimit				:= lrTorqueLimit, 
						LagLimit				:= lrLagLimit, 
						Options					:= stOptions);
				
				nStep							:= 1000;
				
			ELSE

				mcStepBlock(Axis				:= Axis, 
						Parameter				:= stParameter, 
						Execute					:= TRUE, 
						Direction				:= eDirection, 
						Velocity				:= lrVelocity,
						SetPosition				:= lrSetPosition, 
						DetectionVelocityLimit	:= lrDetectionVelocityLimit, 
						DetectionVelocityTime	:= tDetectionVelocityTime, 
						TimeLimit				:= tTimeLimit, 
						DistanceLimit			:= lrDistanceLimit, 
						TorqueLimit				:= lrTorqueLimit, 
						TorqueTolerance			:= lrTorqueTolerance, 
						Options					:= stOptions);
						
				nStep							:= 2000;
				
			END_IF
		END_IF
	
	1000: // Wait till end
	
		IF mcStepBlockLag.Done THEN
			mcStepBlockLag.Execute				:= FALSE;
			nStep 								:= 3000;
		END_IF
		
		IF mcStepBlockLag.CommandAborted THEN
			mcStepBlockLag.Execute				:= FALSE;
			bBusy 								:= FALSE;
			bCommandAborted						:= TRUE;
			nStep 								:= 6000;
		END_IF
		
		IF mcStepBlockLag.Error THEN
			mcStepBlockLag.Execute				:= FALSE;
			udiErrorID_Int						:= mcStepBlockLag.ErrorID;
			nStep 								:= 4000;
		END_IF
	
	2000: // Wait till end
	
		IF mcStepBlock.Done THEN
			mcStepBlock.Execute					:= FALSE;
			nStep 								:= 3000;
		END_IF
		
		IF mcStepBlock.CommandAborted THEN
			mcStepBlock.Execute					:= FALSE;
			bBusy 								:= FALSE;
			bCommandAborted						:= TRUE;
			nStep 								:= 6000;
		END_IF
		
		IF mcStepBlock.Error THEN
			mcStepBlock.Execute					:= FALSE;
			udiErrorID_Int						:= mcStepBlock.ErrorID;
			nStep 								:= 4000;
		END_IF
		
	3000: // MC_FinishHoming
	
		mcFinishHoming.Execute					:= TRUE;				
		nStep									:= nStep + 10;
		
	3010: // Wait till end
	
		IF mcFinishHoming.Done THEN
			mcFinishHoming.Execute				:= FALSE;
			bBusy 								:= FALSE;
			bDone 								:= TRUE;
			nStep 								:= 5000;
		END_IF
		
		IF mcFinishHoming.CommandAborted THEN
			mcFinishHoming.Execute				:= FALSE;
			bBusy 								:= FALSE;
			bCommandAborted						:= TRUE;
			nStep 								:= 6000;
		END_IF
		
		IF mcFinishHoming.Error THEN
			mcFinishHoming.Execute				:= FALSE;
			bBusy 								:= FALSE;
			bError								:= TRUE;
			udiErrorID							:= mcFinishHoming.ErrorID;
			nStep 								:= 10000;
		END_IF	
		
	4000: // MC_AbortHoming
	
		mcAbortHoming.Execute					:= TRUE;				
		nStep									:= nStep + 10;
		
	4010: // Wait till end
	
		// No matter what is the end, we go to error State
		IF NOT mcAbortHoming.Busy THEN
			mcAbortHoming.Execute				:= FALSE;
			bBusy 								:= FALSE;
			bError								:= TRUE;
			udiErrorID							:= udiErrorID_Int;			
			nStep								:= 10000;
		END_IF
		
	5000: // Done
		
		bDone									:= bExecute;
		IF NOT bExecute THEN
			nStep 								:= 0;
		END_IF	
	
	6000: // Command Aborted
	
		bCommandAborted							:= bExecute;
		IF NOT bExecute THEN
			nStep 								:= 0;
		END_IF
		
	10000..20000: // Error
	
		bError									:= bExecute;
		IF NOT bExecute THEN
			udiErrorID							:= 0;
			udiErrorID_Int						:= 0;
			nStep 								:= 0;
		END_IF
		
END_CASE
//===============================================================

END_FUNCTION_BLOCK

// ---- POUs/FB/NewFBs/FB_CatchStationWithSensor.TcPOU
(*
Nazwa:			FB_CatchStation
Opis:			Chwytak pod stacjami 
Wersja:			v1.01
Data:			2025-09-04
Autor:			TW,DP
Urzadzenia:		Silownik chwytania, podnośnik JIESANG
Konfiguracja:	
Zmiany:
- 20250904 [DP] EventLog-do sprawdzenia, 1 spr->wywołać błędy 
Info:
- dodano błędy od nastaw powyżej max i min (error 7 i 8)
- dodawno bHomingNeeded
- wylaczanie wyjść zmiana 2 wylaczanie wyjsc jak zniknie Enable
*)


FUNCTION_BLOCK FB_CatchStationWithSensor
VAR_INPUT
	bEnable											: BOOL;				//Zezwolenie na pracę
	bEStop											: BOOL;				//Stop Awaryjny włączony
	bRun											: BOOL;				//Rozkaz łapania 
	bHoming											: BOOL;				//Zezwolenie na wykonanie bazowania i pozycjonowania podajnika
	bHeightSet										: BOOL;				//Ustaw wysokość
	bChangeover										: BOOL;				//Ustawianie na zadaną wysokość do wymiany elementów formatowych
	
	diSensorMeasurementValue						: DINT;				//IOLink zmienna z czujnika balluff
	lrSensorTolerance								: LREAL;			//Tolerancja czujnika
	lrSensorLowBorder								: LREAL;			//Dolny zakres, Wprowadzam bo mam problem z dozownikiem 1 w UBL50
	bAcceptOpenCalibrationValue						: BOOL;				//Kalibracja. Operator potwierdza że chwytak jest otwarty.
	bAcceptCloseCalibrationValue					: BOOL;				//Kalibracja. Operator potwierdza że chwytak złapał butelkę.
	
	bIgnoreError									: BOOL;				//Ignorowania błędów cyklu pracy
	bReset											: BOOL;				//Reset błędu, jeśli w stanie "eError"
	nPositionHeightSV								: LREAL;			//Wysokość zadana na której ma znajdować się stacja
	
	lrMaxHeight										: LREAL;			//Maksymalna wysokość podnośnika chwytaka
	lrMinHeight										: LREAL;			//Minimalna wysokość podnośnika chwytaka
	bManualMovement									: BOOL;				//Zezwolenie na ruchy ręcznę
	bUnlockColision									: BOOL := FALSE;		//Odblokowywanie możliwośći kolizji
	bAlarmSVCVDiffHeightDisable						: BOOL;				//Wyłączenie alarmu od rożnicy wysokości zadanej od aktualnej
	bNoLifter										: BOOL;				//Podnośnik
	bLongerCatchingTime								: BOOL;
		
	bHeightMotorEncoderPulse 						: BOOL;				//Sygnał impulsów enkodera siłownika
	rHeightMotorPositionOffset 						: REAL;				//Wysokość bazowani podnośnika

	_ALARMINFO_						 				: BOOL;
	iStationIndex									: UDINT;			//Numer stacji 
	sStationName									: WSTRING;			//Nazwa stacji	
	
	_HEIGHTMOTOR_ :BOOL;	
		
    udiHeightMotorEncoderCV		: UDINT;
	bHeightEncoderSetCDone		: BOOL;	
	
END_VAR
VAR_OUTPUT
	eState											: E_Station;				//Stan ogólny bloku
	eRunningState									: E_CatchStationState;		//Stan wewnętrzny
	bWarning										: BOOL;						//Ostrzeżenie
	bError											: BOOL;						//Błąd stacji
	nErrorNr										: UDINT;					//Nr błędu podajnika platynek
	sErrorDescription								: STRING(200);				//Opis błędu
	sErrorDescription2								: STRING(200);				//Opis błędu 2
	sErrorStationName								: STRING;					//Nazwa stacji
	udiStationID									: UDINT;					// Nr stacj
	bCatchActuator									: BOOL;						//Sterownie siłownika łapania opakowania
	
	bHeightMotorUp									: BOOL;						//Sterowanie silnikiem podnośnika  - RUCH W GÓRĘ
	bHeightMotorDown								: BOOL;						//Sterowanie silnikiem podnośnika  - RUCH W DÓŁ
	lrHeightMotorCV									: LREAL;					//Aktualna pozycja podnośnika
	tCycleTime										: TIME;
	bHomingDone										: BOOL;						//Wymagane ponowne bazowanie (blad podczas bazowania lub stop awaryjny)
	bCalibrationDone								: BOOL;						//Potwierdzenie popranej kalibracji czujnika
	bCycleDone										: BOOL;
	bCycleNotDone									: BOOL;
	
	udiHeightMotorEncoderSetCV	: UDINT;		
	bHeightEncoderSetC			: BOOL;	
	
END_VAR
VAR
	tonHeightNoChange								: TON; 						//Timer wykrycia braku ruchu siłownika zmiany wysokości stacji
	nLastPositionHeightCV							: LREAL;					//Pozycja podnośnika w poprzednim cyklu programu
	tonErrorHeightChange							: TON; 						//Timer błędu podnośnika
	
	// Czas zadziałania siłownika
	tonCatchingTime									: TON;
	
	// Timer blokady otwierania chwytaka
	tonOpeningBlocked								: TON;
	tonCycleTimer									: TON;
	rtEncoderHomed									: R_TRIG;
	rtrigCycleTimerRead								: R_TRIG;
	
	tofMotorUpPermition								: TOF;
	tofMotorDownPermition							: TOF;
	tonLimitPosMinReachedDelay						: TON;
	tonLimitPosMaxReachedDelay						: TON;
	tonMaxHeight									: TON;
	tonMinHeight									: TON;
	tonSVCVDiffHeight								: TON;
	
	//Podnośnik Jiesang	
	fbHeightMotorEncoder: FB_JiesangActuatorEncoderModul;	// Blok enkodera podnośnika chwytaka stabilizującego pod zakręcarką	
	bHeightMotorEncoderCounterReset					:BOOL; 							//Sygnał resetu enkodera
	bHeightMotorEncoderHomed						:BOOL;							//Informacja od enkodera że jest zbazowany

	eLastState										: E_Station;					//Stan ogólny bloku
	eLastRunningState								: E_CatchStationState;			//Stan podbloku
	eLastStateTemp									: E_Station;					//Stan ogólny bloku
	eLastRunningStateTemp							: E_CatchStationState;			//Stan podbloku
	bStateError										: BOOL;

	tonStopping										: TON;
	tofHeightMotorDown								: TOF;
	iCaseChangeover									: INT;
	tonChangeOverLimitPosMinReachedDelay			: TON;
	tonChangeoverLimitPosMaxReachedDelay			: TON;
	
	rtAcceptOpenCalibrationValue					: R_TRIG;						//R_TRIG, potwierdzenie otwarcia
	rtAcceptCloseCalibrationValue					: R_TRIG;						//R_TRIG, potwierdzenie zamknięcia
	
	bOpenedActuatorSensor							: BOOL;							//Czujnik otwarcia siłownika łapania
	bClosedActuatorSensor							: BOOL;							//Czujnik otwarcia siłownika łapania
	tonbAcceptCloseCalibrationValue					: TON;
	tonbAcceptOpenCalibrationValue					: TON;
	
	arrNotCatchStatistics							: ARRAY [0..100] OF LREAL;		//Statystyka NOT Catch
	count											: INT;							//Licznik NOT Catch
	bLowBorderActive								: BOOL;							//Załączenie dolnego zakresu
	icoint: INT;
	
		//Zmienne od EVENTLOGGER
	bAlarmInit 						: BOOL := TRUE; 
	nAlarmNumerator					: INT;
	arfbAlarm						: ARRAY[0..19] OF  FB_TcAlarm;		//Tablica bloczków błędów
	fbSourceInfo 					: FB_TcSourceInfo;
	iSourceInfo						: I_TcSourceInfo;
	sAlarmTest						: STRING;
	//Koniec zmiennych od EVENTLOGGER
	bTest							: BOOL;
END_VAR

VAR_IN_OUT
	lrWeighedOpenedValue							: LREAL;						//Zmieżona wartość zamknięcia chwytaków				
	lrWeighedClosedValue							: LREAL;						//Zmieżona wartość zamknięcia chwytaków
	lrMeasuredOpenedValueShow						: LREAL;					//Zmieżona wartość zamknięcia chwytaków				
	lrMeasuredClosedValueShow						: LREAL;					//Zmieżona wartość zamknięcia chwytaków
	bManualCatchActuator							: BOOL;							//Ruch ręczny siłownikiem podajnika platynek
	bManualHeightMotorUp							: BOOL;							//Ruch ręczny podnośnika stacji w górę
	bManualHeightMotorDown							: BOOL;							//Ruch ręczny podnośnika stacji w dół
END_VAR


IF lrSensorLowBorder <> 0 THEN
	bLowBorderActive								:= TRUE;
ELSE
	bLowBorderActive								:= FALSE;
END_IF

Calibration();
HeightMotor();
ErrorHandling();
Control();
Changeover();
Statistics();
aStationID();

(*Zapisywanie ostatniego stanu*)
IF eLastStateTemp<>eState THEN
	eLastState := eLastStateTemp;
END_IF
eLastStateTemp := eState;
IF eLastRunningStateTemp<>eRunningState THEN
	eLastRunningState := eLastRunningStateTemp;
END_IF
eLastRunningStateTemp := eRunningState;
(*Koniec Zapisywanie ostatniego stanu*)


nLastPositionHeightCV:=lrHeightMotorCV;

ACTION aStationID:
udiStationID	:=	iStationIndex;
END_ACTION

ACTION Calibration:
//Najpierw zamyka/otwiera chwytak nastepnie po czasie kalibrje
tonbAcceptCloseCalibrationValue		(IN:=bAcceptCloseCalibrationValue,	PT:=T#2S);
tonbAcceptOpenCalibrationValue		(IN:=bAcceptOpenCalibrationValue,	PT:=T#2S);

rtAcceptCloseCalibrationValue		(CLK:= tonbAcceptCloseCalibrationValue.Q);
rtAcceptOpenCalibrationValue		(CLK:= tonbAcceptOpenCalibrationValue.Q);


IF rtAcceptCloseCalibrationValue.Q THEN
	lrMeasuredClosedValueShow							:= (DINT_TO_LREAL(diSensorMeasurementValue)/1000.0); 
END_IF

IF rtAcceptOpenCalibrationValue.Q THEN
	lrMeasuredOpenedValueShow							:= (DINT_TO_LREAL(diSensorMeasurementValue)/1000.0);
END_IF


IF (lrWeighedClosedValue*1000.0) <> 0 AND (lrWeighedOpenedValue*1000.0) <> 0 THEN
	bCalibrationDone									:= TRUE;
ELSE
	bCalibrationDone									:= FALSE;
END_IF


IF bCalibrationDone THEN
	
	//Chwytak OTWARTY
	IF (diSensorMeasurementValue <= (lrWeighedOpenedValue*1000.0) + lrSensorTolerance) AND (diSensorMeasurementValue >= (lrWeighedOpenedValue*1000.0) - lrSensorTolerance) THEN
		
		bOpenedActuatorSensor							:= TRUE;
	
	ELSE

		bOpenedActuatorSensor							:= FALSE;
	
	END_IF
	
	
	//Chwytak ZAMKNIĘTY
	IF (diSensorMeasurementValue <= (lrWeighedClosedValue*1000.0) + lrSensorTolerance) AND (diSensorMeasurementValue >= (lrWeighedClosedValue*1000.0) - lrSensorTolerance) THEN
	
		bClosedActuatorSensor							:= TRUE;
	
	ELSE
		
		bClosedActuatorSensor							:= FALSE;
	
	END_IF
	
ELSE
	
	bOpenedActuatorSensor								:= FALSE;
	bClosedActuatorSensor								:= FALSE;
	
END_IF
END_ACTION

ACTION Changeover:
tonChangeOverLimitPosMinReachedDelay(IN:=(lrHeightMotorCV<=lrMinHeight) AND bChangeover,PT:=T#2S);
tonChangeoverLimitPosMaxReachedDelay(IN:=(lrHeightMotorCV>=lrMaxHeight) AND bChangeover,PT:=T#2S);


//Przeniesione do PreparingToDisabled
(*CASE iCaseChangeover OF
	
	0: //Włączenie ustawiania
		IF bChangeover THEN
			iCaseChangeover := iCaseChangeover + 10;
			bHeightMotorDown:=FALSE;
			bHeightMotorUp:=FALSE;
		END_IF
		
	10: //Ustawianie stacji na wysokość 
		IF bHeightMotorEncoderHomed THEN
			bHeightMotorEncoderCounterReset	:=	FALSE;
			bHeightMotorUp					:=	lrHeightMotorCV	<=	200;
			bHeightMotorDown				:=	lrHeightMotorCV	>=	200;
			//Kiedy stacja osiągnie wysokość zadaną
			IF ABS(lrHeightMotorCV-nPositionHeightSV)<2 OR tonChangeoverLimitPosMaxReachedDelay.Q OR tonChangeOverLimitPosMinReachedDelay.Q  THEN
				bHeightMotorDown			:=	FALSE;
				bHeightMotorUp				:=	FALSE;
				iCaseChangeover 			:=	iCaseChangeover + 10;
			END_IF			
		ELSE
			bHeightMotorDown		:=	FALSE;
			bHeightMotorUp			:=	FALSE;
			iCaseChangeover 		:=  0;
		END_IF	
		
	20: //Czekanie na wyłączenie przezbrajania i ustawienie na odpowiednią wysokość z receptury
			IF NOT bChangeover THEN
				iCaseChangeover := iCaseChangeover + 10;
			END_IF
	30: //Ustawianie stacji na wysokość z receptury
		IF bHeightMotorEncoderHomed THEN
			bHeightMotorEncoderCounterReset	:=	FALSE;
			bHeightMotorUp					:=	lrHeightMotorCV	<=	nPositionHeightSV;
			bHeightMotorDown				:=	lrHeightMotorCV	>=	nPositionHeightSV;
			//Kiedy stacja osiągnie wysokość zadaną
			IF ABS(lrHeightMotorCV-nPositionHeightSV)<2 OR tonChangeoverLimitPosMaxReachedDelay.Q OR tonChangeOverLimitPosMinReachedDelay.Q  THEN
				bHeightMotorDown			:=	FALSE;
				bHeightMotorUp				:=	FALSE;
				iCaseChangeover 			:=	iCaseChangeover + 10;
			END_IF			
		ELSE
			bHeightMotorDown		:=	FALSE;
			bHeightMotorUp			:=	FALSE;
			iCaseChangeover 		:=  0;
		END_IF
	40: //Ustawianie stacji na wysokość z receptury	
		iCaseChangeover 		:=  0;

END_CASE
*)
END_ACTION

ACTION Control:

	(** TIMERY**)
	rtEncoderHomed(CLK:=bHeightMotorEncoderHomed,Q=>);
	tonHeightNoChange(IN:=((bHeightMotorUp OR bHeightMotorDown) AND (nLastPositionHeightCV=lrHeightMotorCV)), PT:=T#1S); 
	tonLimitPosMinReachedDelay(IN:=(lrHeightMotorCV<=lrMinHeight) AND eState=E_Station.eHoming,PT:=T#2S);
	tonLimitPosMaxReachedDelay(IN:=(lrHeightMotorCV>=lrMaxHeight) AND eState=E_Station.eHoming,PT:=T#2S);
	tonStopping(IN:=eState=E_Station.eStopping,PT:=T#2S);
	tofMotorUpPermition(IN:=bHeightMotorDown,PT:=T#250MS);
	tofMotorDownPermition(IN:=bHeightMotorUp ,PT:=T#250MS);	
	(*****Wyłączenie enable*****)
	IF NOT bEnable OR bChangeover THEN //Lub przezbrajania
		IF eState <> E_Station.eDisabled AND eState <> E_Station.ePreparingToDisable THEN
				eState 				:= E_Station.ePreparingToDisable; 
		END_IF	
	END_IF

	(*****Estop*****)
	IF NOT bEstop  THEN	
		IF eState <> E_Station.eAborted AND eState <> E_Station.eAborting AND eState <> E_Station.eDisabled THEN
				eState 				:= E_Station.eAborting; 
		END_IF
	END_IF

	CASE eState OF
	/////////////////////////////	
		E_Station.eDisabled: 					// Stan nieaktywnosci (Stacja wyłączona) 

			IF bEnable THEN
				eState 				:= E_Station.ePreparingToReady; 
			END_IF 
			
    /////////////////////////////	    
		E_Station.eAborted: 					// Stan bezpiecznego zatrzymania (po Abortingu) 

			IF bEStop THEN
				eState 				:= E_Station.ePreparingToReady;
			END_IF
			
	/////////////////////////////	
		E_Station.eAborting:                 	// Stan bezpiecznego zatrzymywania (po EStopie)

			bHeightMotorUp				:=	FALSE;
			bHeightMotorDown			:=	FALSE;
			eState := E_Station.eAborted;  
			eRunningState:=E_CatchStationState.eDisabled;
			
	/////////////////////////////			
		E_Station.eError:                 	 	// Stan błędu 	

			iCaseChangeover 		:=	0;
			IF bReset THEN
				eState 				:=	E_Station.eResetting;
			END_IF
						
	/////////////////////////////
		E_Station.eResetting:					// Stan resetowania bledu (po Errorze)
	
			bError := FALSE;

			IF NOT bError THEN
				nErrorNr 			:=	0;
   				sErrorDescription 	:=	'';
				eState 				:=	E_Station.ePreparingToReady;
			ELSE
				eState 				:=	E_Station.eError;
			END_IF
        
	/////////////////////////////
		E_Station.eManualMovement:     			// Stan ruchów manualnych  

			ManualMovements();
			//Wyjście z trybu serwisowego
			IF NOT bManualMovement THEN
				bCatchActuator				:=	FALSE;
				bHeightMotorUp				:=	FALSE;
				bHeightMotorDown			:=	FALSE;
				bManualCatchActuator		:=	bCatchActuator;
				eState:=E_Station.eReady;
			END_IF

	/////////////////////////////
		E_Station.eHoming:						// Stan bazowania 

			Homing();
			IF NOT bHoming AND NOT bHeightSet THEN
			   eState:=E_Station.ePreparingToReady;
			   	bHeightMotorDown:=FALSE;
				bHeightMotorUp:=FALSE;
			END_IF		
			
	/////////////////////////////
		E_Station.eHomingDone:                  // Stan wykonania bazowania 
	
			bHeightMotorDown					:=	FALSE;
			bHeightMotorUp						:=	FALSE;
			bHeightMotorEncoderCounterReset		:=	FALSE;
			bHomingDone							:=	TRUE;
			IF NOT bHoming AND NOT bHeightSet THEN
			   eState:=E_Station.eReady;
			END_IF
			
	/////////////////////////////
		E_Station.ePreparingToReady:            // Stan przygotowywania do gotowosci (zawsze przed Ready)  
	
			bCatchActuator	:=	FALSE;
			eRunningState	:=	E_CatchStationState.eReady;
			eState			:=	E_Station.eReady;	
			
	/////////////////////////////
		E_Station.ePreparingToDisable:          // Stan przygotowywania do nieaktywnosci (po wyłączeniu Enable) 
  
			bCatchActuator:=FALSE;
			IF NOT bChangeOver THEN //Normalne wyłączenie
				bHeightMotorUp:=TRUE;
				bHeightMotorDown:=FALSE;	
				IF tonHeightNoChange.Q THEN
					bHeightMotorUp:=FALSE;
					eState:=E_Station.eDisabled;
					eRunningState:=E_CatchStationState.eDisabled;
				END_IF	
			ELSE //Wyłączenie z przebrajaniem na pozycje 200
				IF bHeightMotorEncoderHomed THEN
					bHeightMotorEncoderCounterReset	:=	FALSE;
					bHeightMotorUp					:=	lrHeightMotorCV	<=	150 AND NOT tofMotorUpPermition.Q;
					bHeightMotorDown				:=	lrHeightMotorCV	>=	150 AND NOT tofMotorDownPermition.Q;
					//Kiedy stacja osiągnie wysokość zadaną
					IF ABS(lrHeightMotorCV-150)<2 OR tonChangeoverLimitPosMaxReachedDelay.Q OR tonChangeOverLimitPosMinReachedDelay.Q  THEN
						bHeightMotorDown			:=	FALSE;
						bHeightMotorUp				:=	FALSE;
						eState						:=	E_Station.eDisabled;
						eRunningState				:=	E_CatchStationState.eDisabled;
					END_IF			
				ELSE
					bHeightMotorDown				:=	FALSE;
					bHeightMotorUp					:=	FALSE;
					eState								:=E_Station.eDisabled;
					eRunningState					:=	E_CatchStationState.eDisabled;
				END_IF	
			END_IF
				
	/////////////////////////////
		E_Station.eReady:						// Stan gotowosci 

			IF bRun  AND NOT bCycleDone AND NOT bCycleNotDone THEN
				eState 				:= E_Station.eStarting; 
			END_IF
			IF bHoming OR bHeightSet OR bChangeover THEN
				eState 				:= E_Station.eHoming; 				
			END_IF
			IF bManualMovement THEN
				//Jeśli przejście w tryb ruchów manualnych przepisz wszystkie stany siłowników sterowanych przez moduł
				//aby zapobiec ewentualnym kolizjom po wejściu w tryb serwisowy
				bManualCatchActuator		:= bCatchActuator;
				bManualHeightMotorUp		:= bHeightMotorUp;
				bManualHeightMotorDown		:= bHeightMotorDown;
				
				eState 						:= E_Station.eManualMovement; 
				eRunningState 				:= E_CatchStationState.eReady;
 
			END_IF
			IF NOT bRun THEN
				bCycleDone 			:= FALSE;
				bCycleNotDone 		:= FALSE;			
			END_IF
			
	/////////////////////////////
		E_Station.eStopping:					// Stan zatrzymywania 
					
			Running();
			IF bOpenedActuatorSensor OR tonStopping.Q THEN //NEW
				eState						:=	E_Station.eReady;
				eRunningState 				:=	E_CatchStationState.eReady;
			END_IF
			
	/////////////////////////////
		E_Station.eStarting:                  	// Stan uruchamiania (po Ready)
				
			eState					 := E_Station.eRunning; 

	/////////////////////////////
		E_Station.eRunning:               		// Stan wykonywania cyklu (po Startingu), w tym stanie osobny

			Running();
			IF NOT bRun THEN 					(*Przerywanie cyklu*)
				eState				:= E_Station.eStopping;
				bCycleNotDone		:= TRUE;
			END_IF
			(*IF bCycleDone OR bCycleNotDone THEN (*Cykl zakończony*)
				eState 				 := E_Station.eReady;
			END_IF*)						
		ELSE
		
		
	/////////////////////////////		
	END_CASE
END_ACTION

ACTION ErrorHandling:
// Alarm_0240	240	Error	Blokada otwarcia chwytaka - sprawdź czujnik
// Alarm_0241	241	Error	Blokada podnośnika lub brak zasilania - sprawdź czujnik lub odblokuj mechanicznie
// Alarm_0242	242	Error	Wartość zadana wysokości jest większa od maksymalnej - zmień ustawienia w recepturze {0}
// Alarm_0243	243	Error	Wartość zadana wysokości jest mniejsza od minimalnej - zmień ustawienia w recepturze {0}
// Alarm_0244	244	Error	Wartość aktualna jest zbyt różna od zadanej - zmień ustawienia w recepturze lub ustaw stację
// Alarm_0245	245	Error	Błąd napędu przeciągania. Błąd NC: {0}


IF bAlarmInit THEN
    bAlarmInit := FALSE; 
	fbSourceInfo.Clear();
	fbSourceInfo.sName:=wsLiteral_TO_UTF8(sStationName);//'Machine';
	fbSourceInfo.nId:=iStationIndex;//2700;
	// Alarm_0240	240	Error	Blokada otwarcia chwytaka - sprawdź czujnik
    arfbAlarm[0].CreateEx(stEventEntry := TC_EVENTS.AlarmClass.Alarm_0240, bWithConfirmation:= FALSE,  ipSourceInfo:= fbSourceInfo); 
	// Alarm_0241	241	Error	Blokada podnośnika lub brak zasilania - sprawdź czujnik lub odblokuj mechanicznie
	arfbAlarm[1].CreateEx(stEventEntry := TC_EVENTS.AlarmClass.Alarm_0241, bWithConfirmation:= FALSE,  ipSourceInfo:= fbSourceInfo); 
	// Alarm_0242	242	Error	Wartość zadana wysokości jest większa od maksymalnej - zmień ustawienia w recepturze
	arfbAlarm[2].CreateEx(stEventEntry := TC_EVENTS.AlarmClass.Alarm_0242, bWithConfirmation:= FALSE,  ipSourceInfo:= fbSourceInfo); 
	// Alarm_0243	243	Error	Wartość zadana wysokości jest mniejsza od minimalnej - zmień ustawienia w recepturze
	arfbAlarm[3].CreateEx(stEventEntry := TC_EVENTS.AlarmClass.Alarm_0243, bWithConfirmation:= FALSE,  ipSourceInfo:= fbSourceInfo); 
	// Alarm_0244	244	Error	Wartość aktualna jest zbyt różna od zadanej - zmień ustawienia w recepturze lub ustaw stację
	arfbAlarm[4].CreateEx(stEventEntry := TC_EVENTS.AlarmClass.Alarm_0244, bWithConfirmation:= FALSE,  ipSourceInfo:= fbSourceInfo); 
END_IF


//OBSŁUGA BŁĘDÓW PODAJNIKA PLATYNEK

//************LISTA BŁĘDÓW***************
bStateError:= (eState=E_Station.eError) OR (eState=E_Station.eResetting) OR bIgnoreError;

IF bEnable THEN
	
	//Warning, Kalibracja czujnika
	IF NOT bCalibrationDone THEN
		
		bWarning								:= TRUE;
		sErrorDescription						:= 'Czujnik wymaga kalibracji';
	ELSE
	
		bWarning								:= FALSE;
		sErrorDescription						:= '';
			
	END_IF	

	// Alarm_0240	240	Error	Blokada otwarcia chwytaka - sprawdź czujnik
	//Error 1 - Blokada otwarcia chwytaka
	tonOpeningBlocked(IN:=NOT bCatchActuator AND NOT bOpenedActuatorSensor AND bEStop OR bTest, PT:=T#3S);
	
	IF tonOpeningBlocked.Q AND NOT bWarning THEN
		IF NOT arfbAlarm[0].bActive THEN
			arfbAlarm[0].Raise(nTimeStamp:=0);
		END_IF
	ELSE	
		IF  arfbAlarm[0].bActive AND bReset THEN
			arfbAlarm[0].Clear(nTimeStamp:=0, bResetConfirmation:= FALSE);
		END_IF	
// 		sErrorDescription						:= 'Blokada otwarcia chwytaka - sprawdź czujnik';
// 		bHeightMotorUp							:= FALSE;
// 		bError 									:= TRUE;
// 		nErrorNr								:= 161;	
// 		//nErrorNr 								:= nErrorNr+iStationIndex;
// 		
	END_IF
	
	// Alarm_0241	241	Error	Blokada podnośnika lub brak zasilania - sprawdź czujnik lub odblokuj mechanicznie
	//Error 2 - podnośnik nie porusza się pomimo wysterowania 
	tonErrorHeightChange(IN:=(bHeightMotorUp OR bHeightMotorDown) AND nLastPositionHeightCV=lrHeightMotorCV AND NOT bNoLifter, PT:=T#5S);
	
	IF tonErrorHeightChange.Q THEN
		IF NOT arfbAlarm[1].bActive THEN
			bHeightMotorUp							:= FALSE;
			bHeightMotorDown						:= FALSE;
			arfbAlarm[1].Raise(nTimeStamp:=0);
		END_IF
	ELSE	
		IF  arfbAlarm[1].bActive AND bReset THEN
			arfbAlarm[1].Clear(nTimeStamp:=0, bResetConfirmation:= FALSE);
		END_IF	
// 		bHeightMotorUp							:= FALSE;
// 		bHeightMotorDown						:= FALSE;
// 		bError 									:= TRUE;
// 		nErrorNr								:= 162;
// 		//nErrorNr 								:= nErrorNr+iStationIndex;
// 		sErrorDescription						:= 'Blokada podnośnika lub brak zasilania - sprawdź czujnik lub odblokuj mechanicznie';	
		
	END_IF
	
	// Alarm_0242	242	Error	Wartość zadana wysokości jest większa od maksymalnej - zmień ustawienia w recepturze {0}
	//Error 7 - Bład nastaw max
	tonMaxHeight(IN:=nPositionHeightSV>lrMaxHeight+1 AND bHomingDone AND lrMaxHeight>0 AND eState=E_Station.eReady,PT:=T#30S);
	IF tonMaxHeight.Q THEN
		arfbAlarm[2].ipArguments.Clear() .AddLReal(lrMaxHeight);
		IF NOT arfbAlarm[2].bActive THEN
			bHeightMotorUp							:= FALSE;
			bHeightMotorDown						:= FALSE;
			arfbAlarm[2].Raise(nTimeStamp:=0);
		END_IF
	ELSE	
		IF  arfbAlarm[2].bActive AND bReset THEN
			arfbAlarm[2].Clear(nTimeStamp:=0, bResetConfirmation:= FALSE);
		END_IF	
// 		bHeightMotorUp							:= FALSE;
// 		bHeightMotorDown						:= FALSE;
// 		bError 									:= TRUE;
// 		nErrorNr								:= 163;
// 		//nErrorNr 								:= nErrorNr+iStationIndex;
// 		sErrorDescription						:= 'Wartość zadana wysokości jest większa od maksymalnej - zmień ustawienia w recepturze';
// 		sErrorDescription2						:= REAL_TO_STRING(LREAL_TO_INT(lrMaxHeight));
		
	END_IF
	
	// Alarm_0243	243	Error	Wartość zadana wysokości jest mniejsza od minimalnej - zmień ustawienia w recepturze {0}
	//Error 8 - Bład nastaw min
	tonMinHeight(IN:=nPositionHeightSV<lrMinHeight-1 AND bHomingDone AND lrMinHeight>0 AND eState=E_Station.eReady,PT:=T#30S);
	
	IF tonMinHeight.Q THEN
		arfbAlarm[3].ipArguments.Clear() .AddLReal(lrMinHeight);
		IF NOT arfbAlarm[3].bActive THEN
			bHeightMotorUp							:= FALSE;
			bHeightMotorDown						:= FALSE;
			arfbAlarm[3].Raise(nTimeStamp:=0);
		END_IF
	ELSE	
		IF  arfbAlarm[3].bActive AND bReset THEN
			arfbAlarm[3].Clear(nTimeStamp:=0, bResetConfirmation:= FALSE);
		END_IF	
// 		bHeightMotorUp							:= FALSE;
// 		bHeightMotorDown						:= FALSE;
// 		bError 									:= TRUE;
// 		nErrorNr								:= 164;
// 		//nErrorNr 								:= nErrorNr+iStationIndex;
// 		sErrorDescription						:= 'Wartość zadana wysokości jest mniejsza od minimalnej - zmień ustawienia w recepturze ';
// 		sErrorDescription2						:= REAL_TO_STRING(LREAL_TO_INT(lrMinHeight));
		
	END_IF
	
	// Alarm_0244	244	Error	Wartość aktualna jest zbyt różna od zadanej - zmień ustawienia w recepturze lub ustaw stację
	//Error 9 - Bład zbyt dużej różnicy nastaw
//	tonSVCVDiffHeight(IN:=ABS(nPositionHeightSV-lrHeightMotorCV)>20 AND bHomingDone AND NOT bAlarmSVCVDiffHeightDisable AND eState=E_Station.eReady,PT:=T#3S);
// 	IF tonSVCVDiffHeight.Q AND NOT bStateError THEN
// 		
// 		bHeightMotorUp							:= FALSE;
// 		bHeightMotorDown						:= FALSE;
// 		bError 									:= TRUE;
// 		nErrorNr								:= 165;
// 		//nErrorNr 								:= nErrorNr+iStationIndex;
// 		sErrorDescription						:= 'Wartość aktualna jest zbyt różna od zadanej - zmień ustawienia w recepturze lub ustaw stację';
// 		sErrorDescription2						:= REAL_TO_STRING(LREAL_TO_INT(nPositionHeightSV));
// 		
// 	END_IF
	
	
ELSE
	bError := FALSE;
END_IF

	
//******************PRZEJŚCIE DO eERROR*****************************

IF bError AND NOT bStateError THEN
	IF eLastState = eRunning THEN
		bCycleNotDone := TRUE;
	END_IF
	eState := E_Station.eError;
END_IF

//****************WYŚWIETLANIE STATUSU BLEDU***********************

(*Wyświetlanie błedu na wyjściu*)
bError							:= FALSE;
FOR nAlarmNumerator := 0 TO 19 DO
	bError						:= bError OR arfbAlarm[nAlarmNumerator].bActive;
END_FOR

(*Przepisywanie nazwy stacji*)
sErrorStationName := WSTRING_TO_STRING(sStationName);


//Jezeli nie zbazowane to potrzebne bazowanie
IF NOT bHeightMotorEncoderHomed AND NOT bNoLifter  THEN
	bHomingDone:=FALSE;
END_IF
END_ACTION

ACTION HeightMotor:
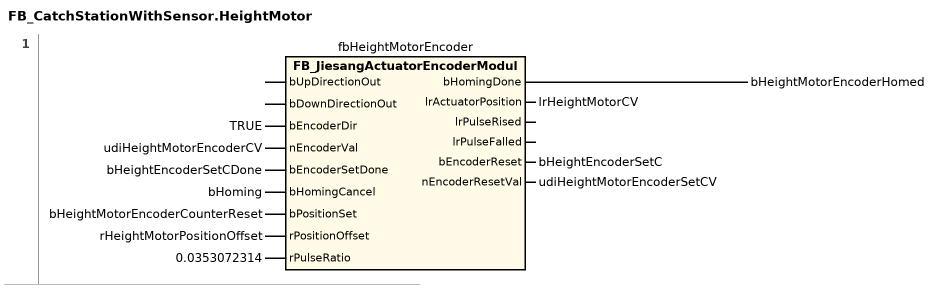
// NETWORK 1
fbHeightMotorEncoder(
    bEncoderDir := TRUE,
    nEncoderVal := udiHeightMotorEncoderCV,
    bEncoderSetDone := bHeightEncoderSetCDone,
    bHomingCancel := bHoming,
    bPositionSet := bHeightMotorEncoderCounterReset,
    rPositionOffset := rHeightMotorPositionOffset,
    rPulseRatio := 0.0353072314,
    lrActuatorPosition => lrHeightMotorCV,
    bEncoderReset => bHeightEncoderSetC,
    nEncoderResetVal => udiHeightMotorEncoderSetCV); // FB_JiesangActuatorEncoderModul
bHeightMotorEncoderHomed := fbHeightMotorEncoder.bHomingDone;
END_ACTION

ACTION Homing:
//BAZOWANIE
bCatchActuator:=FALSE;
	
//Uwaga nie zmieniać czasu bo jednocześnie dwie stację jadą do góry
tofHeightMotorDown(IN:=bHeightMotorDown, PT:=T#1S); //Zabezpieczenie przed zbyt szybkim przełączeniem pomiędzy Down a Up, bezpiecznieki sie palą, 


//Podnoszenie stacji do maksymalnej pozycji
IF NOT bHeightMotorEncoderHomed OR rtEncoderHomed.Q THEN
	bHeightMotorUp:=(*TRUE*) NOT tofHeightMotorDown.Q;;
	bHeightMotorDown:=FALSE;
	IF tonHeightNoChange.Q THEN
		bHeightMotorEncoderCounterReset:=TRUE;
		bHeightMotorUp:=FALSE;
	END_IF
	//Jesli enkoder zbazowany zakończ bazowanie	
	IF rtEncoderHomed.Q THEN
		bHeightMotorUp:=FALSE;
		bHeightMotorDown:=FALSE;
		eState:=E_Station.eHomingDone;
	END_IF		
		
//Po podniesieniu stacji opuszczanie do ustalonej wysokości
ELSIF bHeightMotorEncoderHomed THEN
	bHeightMotorEncoderCounterReset:=FALSE;
	bHeightMotorUp:=lrHeightMotorCV<=nPositionHeightSV;
	bHeightMotorDown:=lrHeightMotorCV>=nPositionHeightSV (*AND lrHeightMotorCV>=lrMinHeight*);
	//Kiedy stacja osiągnie wysokość zadaną
	IF ABS(lrHeightMotorCV-nPositionHeightSV)<1 OR tonLimitPosMaxReachedDelay.Q OR tonLimitPosMinReachedDelay.Q (*OR lrHeightMotorCV>=lrMinHeight*) THEN
		bHeightMotorDown:=FALSE;
		bHeightMotorUp:=FALSE;
		eState:=E_Station.eHomingDone;
	END_IF			
END_IF

	
//Opcja braku podnośnika	
IF bNoLifter THEN
	eState:=E_Station.eHomingDone;
END_IF
END_ACTION

ACTION ManualMovements:

//W trybie ruchów manualnych wykonuj ruchy za pomocą rozkazów manualnych
IF NOT bRun THEN
	bCatchActuator:=bManualCatchActuator;
	IF bAcceptCloseCalibrationValue THEN
		bCatchActuator := TRUE;
	END_IF
	IF bAcceptOpenCalibrationValue THEN
		bCatchActuator := FALSE;;
	END_IF	
	bHeightMotorUp:=bManualHeightMotorUp;
	bHeightMotorDown:=bManualHeightMotorDown;
ELSE	//Kasuje zeby po cyklu nic sie nie poruszało
	bManualCatchActuator := FALSE;
	bManualHeightMotorUp  := FALSE;
	bManualHeightMotorDown  := FALSE;
END_IF


IF bHoming OR bHeightSet THEN
	eState:=E_Station.eHoming;
END_IF
	
Running();
	
//Zabezpieczenie przed kolizją stacji poprzez ruch podnośnika	
IF bHeightMotorDown AND lrHeightMotorCV<=lrMinHeight AND NOT bHoming AND NOT bHeightSet THEN
	bHeightMotorDown:=FALSE;
END_IF	

IF bHeightMotorUp AND lrHeightMotorCV>=lrMaxHeight AND NOT bHoming AND NOT bHeightSet THEN
	bHeightMotorUp:=FALSE;
END_IF		 

IF NOT bRun THEN
	bCycleDone 					:= FALSE;
	bCycleNotDone 				:= FALSE;	
END_IF
END_ACTION

ACTION Running:
//Timery
IF NOT bLongerCatchingTime THEN
	tonCatchingTime(IN:=(eRunningState=E_CatchStationState.eCatching), PT:=T#500MS); //bylo 300
ELSE
	tonCatchingTime(IN:=(eRunningState=E_CatchStationState.eCatching), PT:=T#1100MS); //bylo 300	
END_IF

CASE eRunningState OF
	
	//NIEGOTOWY
	E_CatchStationState.eDisabled:
	
		eRunningState											:= E_CatchStationState.eReady;

		
	//Chwytak gotowy do pracy
	E_CatchStationState.eReady: 
	
		//Jeśli komenda chwytania przejdz do stanu chwytanie
		IF NOT bCycleDone AND NOT bCycleNotDone THEN
			
			IF bRun THEN
				eRunningState									:= E_CatchStationState.eCatching;
			END_IF
			
		END_IF
		
	//Chwytanie 
	E_CatchStationState.eCatching:
	
		bCatchActuator:=TRUE;
		
		IF tonCatchingTime.Q THEN
			
			IF bClosedActuatorSensor OR bLowBorderActive THEN
				eRunningState									:= E_CatchStationState.eCatched;
			ELSE
				arrNotCatchStatistics[count]					:= diSensorMeasurementValue;
				count											:= count + 1;
				eRunningState									:= E_CatchStationState.eNotCatched;
			END_IF
			
		END_IF

	//Uchwycone 
	E_CatchStationState.eCatched:
	
		bCatchActuator											:= bRun;
		bCycleDone 												:= TRUE;
		//Kiedy zniknie rozkaz chwytania i 
	
	E_CatchStationState.eNotCatched:
	
		bCatchActuator											:= bRun;                                   
		bCycleDone 												:= TRUE;
	
END_CASE

IF count  = 100 THEN
	FOR icoint:= 0 TO 100 DO
		arrNotCatchStatistics[icoint]					:= 0;
	END_FOR
	count												:= 0;
END_IF
END_ACTION

ACTION Statistics:



rtrigCycleTimerRead(CLK:=eRunningState=E_CatchStationState.eCatched);
IF rtrigCycleTimerRead.Q THEN
	tCycleTime:=tonCycleTimer.ET;
END_IF
tonCycleTimer(IN:=eState>E_Station.eReady,PT:=T#1D);
END_ACTION

END_FUNCTION_BLOCK

// ---- POUs/FB/FB_EntranceGatesServo.TcPOU
(*
Nazwa:			FB_EntranceGatesFesto
Opis:			Stacja szlabanów do przesuwania formatek	
Wersja:			v1.1
Data:			2020-09-30
Autor:			DP
Urzadzenia:		do 1 szlabanu na siłowniku beckhoff i 1 szlabanu zatrzymującego na końcu
Konfiguracja:	
Info: 
*)
FUNCTION_BLOCK FB_EntranceGatesServo
VAR_INPUT
	bEnable						:BOOL;			//Zezwolenie na pracę
	bEStop						:BOOL;			//Stop Awaryjny włączony
	bRunPrepare					:BOOL;			//Rozkaz przesuwania formatek do środka 
	bRun						:BOOL;			//Rozkaz wpuszczenia dwóch formatek 
	bHoming						:BOOL;			//Zezwolenie na wykonanie bazowania i pozycjonowania podajnika
	bHeightSet					:BOOL;			//Ustaw wysokość
	bIgnoreError				:BOOL;			//Ignorowania błędów cyklu pracy
	bReset						:BOOL;			//Reset błędu, jeśli w stanie "eError"
	bBlocking					:BOOL;			//Blokowanie pierwszego szlabanu

	bOpenedGate1ActuatorSensor	:BOOL;			//Czujnik otwarcia siłownika szlabanu 1
	bOpenedGate2ActuatorSensor	:BOOL;			//Czujnik otwarcia siłownika szlabanu 2
	bClosedGate1ActuatorSensor	:BOOL;			//Czujnik zamknięcia siłownika szlabanu 1
	bClosedGate2ActuatorSensor	:BOOL;			//Czujnik zamknięcia siłownika szlabanu 2
	bMovingTwoForms				:BOOL;			//Przesuwanie o dwie formatki
	bMovingThreeForms			:BOOL;			//Przesuwanie o trzy formatki
	bManualMovement				:BOOL;			//Zezwolenie na ruchy ręcznę
	bHomingStateGate1			:BOOL;			//Stan bazowania szlabanów nr 1
	bHomingStateGate2			:BOOL;			//Stan bazowania szlabanów nr 2
	bResetState					:BOOL;			//Resetowanie stanu stacji

	//Parametry przeciągania formatek

	lrPullReadyPosition			:LREAL;			//Pozycja przeciągania przy starcie dozowania
	lrPullStopOnePhasePosition	:LREAL;			//Pozycja stopu przeciągania przy dozowaniu jednofazowym
	lrPullStopTwoPhasePosition	:LREAL;			//Pozycja stopu przeciągania przy dozowaniu dwufazowym
	lrPullVelocity				:LREAL;			//Prędkość przeciągania 
	lrPullAcceleration			:LREAL;			//Przyśpieszenie przeciągania
	lrPullDeceleration			:LREAL;			//Zwalnianie przeciągania
	
	_ALARMINFO_					:BOOL;
	iStationIndex				:UDINT;			//Numer stacji 
	sStationName				:STRING;		//Nazwa stacji

END_VAR
VAR_OUTPUT
	
	eState						:E_Station;				//Stan ogólny bloku
	eRunningState				:E_EntranceGatesState;	//Stan szlabanów
	bError						:BOOL;					//Błąd stacji	
	nErrorNr					:UDINT;					//Nr błędu podajnika platynek
	sErrorDescription			:STRING(200);			//Opis błędu
	sErrorDescription2			:STRING(200);			//Opis błędu
	sErrorStationName			:STRING;				//Nazwa stacji
	bGate1Actuator				:BOOL;					//Sterownie siłownika szlabanu 1
	bGate2Actuator				:BOOL;					//Sterownie siłownika szlabanu 2
	tCycleTime					:TIME;
	bHomingDone					:BOOL;					//Wymagane ponowne bazowanie (blad podczas bazowania lub stop awaryjny)
	bCyclePrepareDone			:BOOL;
	bCycleDone					:BOOL;
	bCycleNotDone				:BOOL;
	//WEJSCIA WYJSCIA SPRZETOWE
	nPullServoErrorNr			:UDINT;
	lrPullActualPosition		:LREAL;

END_VAR

VAR

	(**********BECKHOFF PRZECIAGANIE******************)
	mcPullMoveAbsolute			:MC_MoveAbsolute; 	// Blok nr 1 ruchu absolutnego tłoka dozownika
	mcPullManualMove			:MC_JOG;			// Blok ruchu manualnego tłokiem dozownika
	mcPullStop					:MC_Stop;			// Blok zatrzymania tłoka dozownika, jeśli to konieczne
	mcPullSoftReset				:MC_Reset;			// Blok łagodnego resetu serwa tloka dozownika
	mcPullPower					:Mc_Power;			// Blok zasilania serwa dozownika
	bPullServoPower				:BOOL; 				// Zalaczenie zasilania serwa
	// Blok resetowania twardego błędu
	fbPullHardReset				:FB_SoEReset;
	bStopped					:BOOL;
		
	// Timer blokady otwierania chwytaka
	tonOpeningGate1Blocked		:TON;
	tonOpeningGate2Blocked		:TON;
	tonClosingGate1Blocked		:TON;
	tonClosingGate2Blocked		:TON;
	tonCycleTimer				:TON;
	rtrigCycleTimerRead			:R_TRIG;	
	bLastStateGate1Actuator		:BOOL;
	bLastStateGate2Actuator		:BOOL;	
	eLastState					:E_Station;				//Stan ogólny bloku
	eLastRunningState			:E_EntranceGatesState;	//Stan podbloku
	eLastStateTemp				:E_Station;				//Stan ogólny bloku
	eLastRunningStateTemp		:E_EntranceGatesState;	//Stan podbloku

	bStateError: BOOL;
		rtPulling: R_TRIG;
	rtPreparingToReady: R_TRIG;
	rtPullingToMiddle: R_TRIG;
	tonDelayServoOn			: TON;

	bNotPreapreToReadyAfterEstop: BOOL;
	lrtest: LREAL;
	tonGate1Actuator: TON;
END_VAR

VAR_IN_OUT
	bManualGate1Actuator	:BOOL;			//Ruch ręczny siłownikiem szlabanu 1
	bManualGate2Actuator	:BOOL;			//Ruch ręczny siłownikiem szlabanu 2
	bManualPullLeft			:BOOL;			//Ruch ręczny przeciąganiem w lewo
	bManualPullRight		:BOOL;			//Ruch ręczny przeciąganiem w prawo
	PullAxisRef				:AXIS_REF;		//Struktura sterowania NC dla serwa zakręcania
END_VAR

(*Przepisywanie Homingu , rozdzielenie wyjść*)

ErrorHandling();
Control();
GatesControlBlocks();
Statistics();


(*wypracowanie sygnałów wyjściowych z bloku*)
lrPullActualPosition:=PullAxisRef.NcToPlc.ActPos;	//Pozycja 


(*Zapisywanie ostatniego stanu*)
IF eLastStateTemp<>eState THEN
	eLastState := eLastStateTemp;
END_IF
eLastStateTemp := eState;
IF eLastRunningStateTemp<>eRunningState THEN
	eLastRunningState := eLastRunningStateTemp;
END_IF
eLastRunningStateTemp := eRunningState;

(*Koniec Zapisywanie ostatniego stanu*)



IF bResetState AND NOT bBlocking THEN
	eState:=E_Station.eReady;
	eRunningState:=eLastRunningState:=E_EntranceGatesState.eReady;
	bGate1Actuator:=bHomingStateGate1;
	bGate2Actuator:=bHomingStateGate2;
END_IF

ACTION Control:

	(** TIMERY**)
	rtPulling(CLK:=eRunningState=E_EntranceGatesState.ePulling AND bOpenedGate1ActuatorSensor AND bClosedGate2ActuatorSensor, Q=>);
	rtPullingToMiddle(CLK:=eRunningState=E_EntranceGatesState.ePullingToMiddle AND bOpenedGate1ActuatorSensor AND bClosedGate2ActuatorSensor, Q=>);
	rtPreparingToReady(CLK:=eRunningState=E_EntranceGatesState.ePreparingToReady AND bClosedGate1ActuatorSensor, Q=>);
	
	tonDelayServoOn(IN:=(eState = E_Station.ePreparingToReady), PT:=T#1200MS);
	tonGate1Actuator(IN:=bGate1Actuator, PT:=T#100MS); // Opóżnienie sygnału wyjścia pierwszego szlabany, uzyte do opoznienia wylaczania drugiego
	(*****Wyłączenie enable*****)
	IF NOT bEnable THEN
		IF eState <> E_Station.eDisabled AND eState <> E_Station.ePreparingToDisable THEN
				eState 				:= E_Station.ePreparingToDisable; 
		END_IF	
	END_IF

	(*****Estop*****)
	IF NOT bEstop  THEN	
		IF eState <> E_Station.eAborted AND eState <> E_Station.eAborting AND eState <> E_Station.eDisabled THEN
				eState 				:= E_Station.eAborting; 
		END_IF
	END_IF

	
	CASE eState OF
	/////////////////////////////	
		E_Station.eDisabled: 					// Stan nieaktywnosci (Stacja wyłączona) 
		
			IF bEnable THEN
				eState 				:= E_Station.ePreparingToReady; 
			END_IF 
			
    /////////////////////////////	    
		E_Station.eAborted: 					// Stan bezpiecznego zatrzymania (po Abortingu) 

			IF bEStop THEN
				eState 				:= E_Station.ePreparingToReady;
			END_IF
			
	/////////////////////////////	
		E_Station.eAborting:                 	// Stan bezpiecznego zatrzymywania (po EStopie)

		mcPullManualMove.JogBackwards		:=	FALSE;
		mcPullManualMove.JogForward			:=	FALSE;
		mcPullMoveAbsolute.Execute 			:=	FALSE;
		
		//bPullServoPower						:=	TRUE;
		mcPullPower.Override				:=	100;		
		mcPullStop.Execute					:=	NOT bStopped;
		bNotPreapreToReadyAfterEstop		:= TRUE;
		IF (mcPullStop.Done OR mcPullStop.Error OR bStopped) THEN
			bStopped						:=	FALSE;
			bPullServoPower					:=	FALSE;
			mcPullStop.Execute				:=	FALSE;
			eLastRunningState				:=	eRunningState;
			eRunningState					:= E_EntranceGatesState.eReady;
			eState 							:=	E_Station.eAborted; 
		END_IF
			
	/////////////////////////////			
		E_Station.eError:                 	 	// Stan błędu 	
	
			mcPullMoveAbsolute.Execute 			:=	FALSE;
			mcPullStop.Execute					:= FALSE;
			IF bReset THEN
				eState 							:=	E_Station.eResetting;
			ELSE
				mcPullSoftReset	(Execute:=FALSE,Axis:=PullAxisRef);		
			END_IF
			
	/////////////////////////////
		E_Station.eResetting:					// Stan resetowania bledu (po Errorze)
			
			//Procedura obsługi resetu w zależności od błędu
			CASE nErrorNr-iStationIndex OF
		
				//Error 1 - ZACIETY SZLABAN
				1:
					bGate1Actuator								:=	FALSE;		
					nErrorNr									:=	0;
					bError										:=	FALSE;
					sErrorDescription							:=	'';		
					
				//Error 8 - SZLABANYW ZŁEJ POZYCJI			
				8: 
					bGate1Actuator								:=	FALSE;		
					bGate2Actuator								:=	TRUE;		// z 17.11.2020
				//IF tonDelayServoOn.Q THEN
					bPullServoPower								:=	TRUE;
				//END_IF
					IF bClosedGate1ActuatorSensor AND mcPullPower.Status THEN	
						mcPullMoveAbsolute.Velocity			:= lrPullVelocity;
						mcPullMoveAbsolute.Position			:= lrPullReadyPosition;
						mcPullMoveAbsolute.Acceleration		:= 15000;
						mcPullMoveAbsolute.Deceleration		:= 15000;
						mcPullMoveAbsolute.Execute			:= TRUE;
					
						//Wykonano ruch
						IF mcPullMoveAbsolute.Done THEN
							mcPullMoveAbsolute.Execute 		:=	FALSE;
							bError := FALSE;
						END_IF		
					END_IF
				//Error 9, Error 10 - BŁĄD SERWA PRZECIAGANIA
				9,10:	
					fbPullHardReset(Execute:=NOT mcPullMoveAbsolute.Execute,Axis:=PullAxisRef);
					mcPullSoftReset(Execute:=TRUE,Axis:=PullAxisRef);																		
					(*IF NOT fbPullHardReset.Busy AND NOT mcPullSoftReset.Busy AND mcPullPower.Status AND NOT PullAxisRef.Status.Error THEN
						fbPullHardReset(Execute:=FALSE,Axis:=PullAxisRef);
						mcPullSoftReset(Execute:=FALSE,Axis:=PullAxisRef);
						mcPullMoveAbsolute.Execute:=TRUE;
						mcPullMoveAbsolute.Position:=lrPullReadyPosition; 
						IF mcPullMoveAbsolute.Done=TRUE THEN
							mcPullMoveAbsolute.Execute:=FALSE;
							nErrorNr:=0;
							nPullServoErrorNr:=0;
							mcPullPower.Override:=100;
							bError := FALSE;
							sErrorDescription:='';	
						END_IF*)
					IF NOT fbPullHardReset.Busy AND NOT mcPullSoftReset.Busy (*AND NOT mcPullPower.Status*) AND NOT PullAxisRef.Status.Error  THEN
						fbPullHardReset(Execute:=FALSE,Axis:=PullAxisRef);
						mcPullSoftReset(Execute:=FALSE,Axis:=PullAxisRef);
						nPullServoErrorNr:=0;
						nErrorNr:=0;
						mcPullPower.Override:=100;
						bError := FALSE;
						sErrorDescription:='';			  	
					END_IF
					
				ELSE
					bError := FALSE;	
	
				END_CASE	
			
			IF NOT bError THEN
				nErrorNr 			:=	0;
   				sErrorDescription 	:=	'';
   				sErrorDescription2 	:=	'';	
				eState 				:=	E_Station.ePreparingToReady;
			ELSE
				eState 				:=	E_Station.eError;
			END_IF
        
	/////////////////////////////
		E_Station.eManualMovement:     			// Stan ruchów manualnych  
       
			ManualMovements();
			//Wyjście z trybu serwisowego
			IF NOT bManualMovement THEN
				
				bGate1Actuator:=bLastStateGate1Actuator;
				bGate2Actuator:=bLastStateGate2Actuator;
	
				//Ruch 
				mcPullPower.Override				:= 100;
				mcPullMoveAbsolute.Velocity			:= lrPullVelocity;
				mcPullMoveAbsolute.Position			:= lrPullReadyPosition;
				mcPullMoveAbsolute.Acceleration		:= 1000;
				mcPullMoveAbsolute.Deceleration		:= 1000;
				mcPullMoveAbsolute.Execute			:= TRUE;
			
				//Wykonano ruch
				IF mcPullMoveAbsolute.Done THEN
					mcPullMoveAbsolute.Execute 		:=	FALSE;
					eState							:=	E_Station.eReady;
					eRunningState					:=	E_EntranceGatesState.eReady;
				END_IF
				
			END_IF

	/////////////////////////////
		E_Station.eHoming:						// Stan bazowania 

			Homing();
			IF NOT bHoming AND NOT bHeightSet THEN
			   eState							:=	E_Station.ePreparingToReady;
			   mcPullManualMove.JogForward		:=	FALSE;
			   mcPullManualMove.JogBackwards	:=	FALSE;
			END_IF		
			
	/////////////////////////////
		E_Station.eHomingDone:                  // Stan wykonania bazowania 
		
			mcPullManualMove.JogForward			:=	FALSE;
			mcPullManualMove.JogBackwards		:=	FALSE;
			bHomingDone							:=	TRUE;
			IF NOT bHoming AND NOT bHeightSet THEN
			   eState:=E_Station.eReady;
			END_IF
			
	/////////////////////////////
		E_Station.ePreparingToReady:            // Stan przygotowywania do gotowosci (zawsze przed Ready)  
		
		eRunningState						:=	E_EntranceGatesState.eReady;
		IF NOT bNotPreapreToReadyAfterEstop THEN //LastRunningState przypisuje w abborting
			bGate1Actuator								:=	FALSE;		
			bGate2Actuator								:=	TRUE;		// z 17.11.2020
			IF tonDelayServoOn.Q THEN
				bPullServoPower								:=	TRUE;
			END_IF
			IF bClosedGate1ActuatorSensor AND mcPullPower.Status THEN
				IF bHomingDone THEN		
					mcPullMoveAbsolute.Velocity			:= lrPullVelocity;
					mcPullMoveAbsolute.Position			:= lrPullReadyPosition;
					mcPullMoveAbsolute.Acceleration		:= 15000;
					mcPullMoveAbsolute.Deceleration		:= 15000;
					mcPullMoveAbsolute.Execute			:= TRUE;
				
					//Wykonano ruch
					IF mcPullMoveAbsolute.Done THEN
						mcPullMoveAbsolute.Execute 		:=	FALSE;
						eRunningState					:=	E_EntranceGatesState.eReady;
						eState							:=	E_Station.eReady;	
					END_IF
								
				ELSIF NOT bHomingDone THEN
					eRunningState						:=	E_EntranceGatesState.eReady;
					eState								:=	E_Station.eReady;	
				END_IF
			END_IF
		ELSE //estop byl trakcie
			IF tonDelayServoOn.Q THEN
				bPullServoPower								:=	TRUE;
			END_IF
			IF  mcPullPower.Status THEN
				//bNotPreapreToReadyAfterEstop				:= FALSE;
				eState										:=	E_Station.eReady;	
				//eRunningState								:=	eLastRunningState; //Wpisze ostatni stan
			END_IF
		END_IF
			
	/////////////////////////////
		E_Station.ePreparingToDisable:          // Stan przygotowywania do nieaktywnosci (po wyłączeniu Enable) 
  
			bGate1Actuator							:=	FALSE;		
			bGate2Actuator							:=	FALSE;		
			bPullServoPower							:=	TRUE;
			
			IF mcPullPower.Status THEN
				mcPullPower.Override				:=	10;
				mcPullMoveAbsolute.Velocity			:=	100;
				mcPullMoveAbsolute.Execute			:=	TRUE;
				mcPullMoveAbsolute.Position			:=	lrPullReadyPosition;
				IF mcPullMoveAbsolute.Done THEN
					mcPullMoveAbsolute.Execute 		:=	FALSE;
					eState							:=	E_Station.eDisabled;
					eRunningState					:=	E_EntranceGatesState.eReady;
				END_IF	
			END_IF
			
			IF bIgnoreError THEN
				eState								:=	E_Station.eDisabled;
				eRunningState						:=	E_EntranceGatesState.eDisabled;
			END_IF
			
	/////////////////////////////
		E_Station.eReady:						// Stan gotowosci 
		
			IF (bRunPrepare OR bRun) AND NOT bCycleDone AND NOT bCycleNotDone THEN
				eState 				:= E_Station.eStarting; 
			END_IF
			IF bHoming OR bHeightSet THEN
				eState 				:= E_Station.eHoming; 
			END_IF
			IF bManualMovement THEN
				//Jeśli przejście w tryb ruchów manualnych przepisz wszystkie stany siłowników sterowanych przez moduł
				//aby zapobiec ewentualnym kolizjom po wejściu w tryb serwisowy
				bLastStateGate1Actuator		:=	bGate1Actuator;
				bLastStateGate2Actuator		:=	bGate2Actuator;
				bManualGate1Actuator		:=	bGate1Actuator;
				bManualGate2Actuator		:=	bGate2Actuator;				
				eState 						:=	E_Station.eManualMovement; 
			END_IF
			IF NOT bRun THEN
				bCycleDone 					:= FALSE;
				bCycleNotDone 				:= FALSE;	
				bCyclePrepareDone			:= FALSE;		
			END_IF
			
			bStopped						:= FALSE;
			mcPullStop.Execute				:= FALSE;
			
	/////////////////////////////
		E_Station.eStopping:					// Stan zatrzymywania 


			Running();		
			
			mcPullStop.Execute				:=	NOT bStopped;

			IF (mcPullStop.Done OR mcPullStop.CommandAborted) THEN
				 bStopped					:=	TRUE;
			END_IF
			
			IF bStopped AND NOT mcPullStop.Execute THEN
				eState 						:=	E_Station.eReady;	
			END_IF
			

	/////////////////////////////
		E_Station.eStarting:                  	// Stan uruchamiania (po Ready)
		
			eState					 := E_Station.eRunning; 
			
	/////////////////////////////
		E_Station.eRunning:               		// Stan wykonywania cyklu (po Startingu), w tym stanie osobny
 
			IF 	bNotPreapreToReadyAfterEstop THEN //Zmiana 17112020
				bNotPreapreToReadyAfterEstop := FALSE;
				eRunningState								:=	eLastRunningState; //Wpisze ostatni stan
			END_IF
		
			Running();
			IF NOT bRun AND NOT bRunPrepare THEN					(*Przerywanie cyklu*)
				eState 				 := E_Station.eStopping;	
			END_IF
			IF bCycleDone OR bCycleNotDone THEN (*Cykl zakończony*)
				//eState 				 := E_Station.eReady;//Zmiana
				eState 				 := E_Station.ePreparingToReady;
			END_IF	
			
	/////////////////////////////		
	END_CASE
END_ACTION

ACTION ErrorHandling:
//OBSŁUGA BŁĘDÓW PODAJNIKA PLATYNEK

//************LISTA BŁĘDÓW***************
bStateError:= (eState=E_Station.eError) OR (eState=E_Station.eResetting);

IF bEnable THEN

	//Error 1 - Blokada otwarcia szlabanu wejściowego nr 1
	tonOpeningGate1Blocked(IN:= bGate1Actuator AND NOT bOpenedGate1ActuatorSensor, PT:=T#2S);
	IF tonOpeningGate1Blocked.Q AND NOT bStateError THEN
		sErrorDescription:='Blokada otwarcia szlabanu wjazdowego nr 1 - sprawdź czujnik lub odblokuj mechanicznie';
		bError := TRUE;
		nErrorNr:=1;	
		nErrorNr:=nErrorNr+iStationIndex;
	END_IF
	
	//Error 2 - Blokada otwarcia szlabanu wejściowego nr 2
	tonOpeningGate2Blocked(IN:= bGate2Actuator AND NOT bOpenedGate2ActuatorSensor, PT:=T#2S);
	IF tonOpeningGate2Blocked.Q AND NOT bStateError THEN
		sErrorDescription:='Blokada otwarcia szlabanu wjazdowego nr 2 - sprawdź czujnik lub odblokuj mechanicznie';
		bError := TRUE;
		nErrorNr:=2;	
		nErrorNr:=nErrorNr+iStationIndex;
	END_IF
				
	//Error 4 - Blokada zamknięcia szlabanu wejściowego nr 1
	tonClosingGate1Blocked(IN:= NOT bGate1Actuator AND NOT bClosedGate1ActuatorSensor, PT:=T#2S);
	IF tonClosingGate1Blocked.Q AND NOT bStateError THEN
		sErrorDescription:='Blokada zamknięcia szlabanu wjazdowego nr 1 - sprawdź czujnik lub odblokuj mechanicznie';
		bError := TRUE;
		nErrorNr:=2;	
		nErrorNr:=nErrorNr+iStationIndex;
	END_IF

	//Error 5 - Blokada zamknięcia szlabanu wejściowego nr 2
	tonClosingGate2Blocked(IN:= NOT bGate2Actuator AND NOT bClosedGate2ActuatorSensor, PT:=T#2S);
	IF tonClosingGate2Blocked.Q AND NOT bStateError THEN
		sErrorDescription:='Blokada zamknięcia szlabanu wjazdowego nr 2 - sprawdź czujnik lub odblokuj mechanicznie';
		bError := TRUE;
		nErrorNr:=2;	
		nErrorNr:=nErrorNr+iStationIndex;
	END_IF	
		
(*	//Error 8 - SZLABANY W ZŁEJ POZYCJI
	IF (ABS(PullAxisRef.NcToPlc.ActPos) - lrPullReadyPosition) > 5 AND bHomingDone AND eState = E_Station.eReady AND NOT bResetState AND NOT bStateError THEN
		bError := TRUE;
		nErrorNr:=8;
		nErrorNr:=nErrorNr+iStationIndex;
		nPullServoErrorNr:=PullAxisRef.Status.ErrorID;
		sErrorDescription:='Szlabany w złej pozycji, zresetuj';
		sErrorDescription2:=INT_TO_STRING(LREAL_TO_INT(PullAxisRef.NcToPlc.ActPos));
	END_IF;	*)
	
	//Error 9 - BŁĄD SERWA PODNOSZENIA ZAKRĘCARKI
	IF (PullAxisRef.Status.Error OR mcPullPower.Error) AND NOT bStateError THEN
		bError := TRUE;
		nErrorNr:=9;
		nErrorNr:=nErrorNr+iStationIndex;
		nPullServoErrorNr:=PullAxisRef.Status.ErrorID;
		sErrorDescription:='Błąd napędu przeciągania Błąd NC:';
		sErrorDescription2:=F_AxErrMsg(nPullServoErrorNr);
	END_IF;	
	
	//Error 10 - BŁĄD INNY SERWA PODNOSZENIA ZAKRĘCARKI
	IF  mcPullMoveAbsolute.Error AND NOT bStateError THEN
		bError := TRUE;
		nErrorNr:=10;
		nErrorNr:=nErrorNr+iStationIndex;
		nPullServoErrorNr:=mcPullMoveAbsolute.ErrorID;
		sErrorDescription:='Błąd napędu przeciągania Błąd NC:';
		sErrorDescription2:=F_AxErrMsg(nPullServoErrorNr);
	END_IF;
	
	
	
ELSE
	bError := FALSE;
END_IF
	
//*******KONIEC LISTA BŁĘDÓW***************	

	

//******************PRZEJŚCIE DO eERROR*****************************

IF bError AND NOT bStateError THEN
	IF eLastState = eRunning THEN
		bCycleNotDone := TRUE;
	END_IF
	eState := E_Station.eError;
END_IF

//****************WYŚWIETLANIE STATUSU BLEDU***********************


(*Wyświetlanie błedu na wyjściu*)
bError;

(*Przepisywanie nazwy stacji*)
sErrorStationName:=sStationName;
END_ACTION

ACTION GatesControlBlocks:
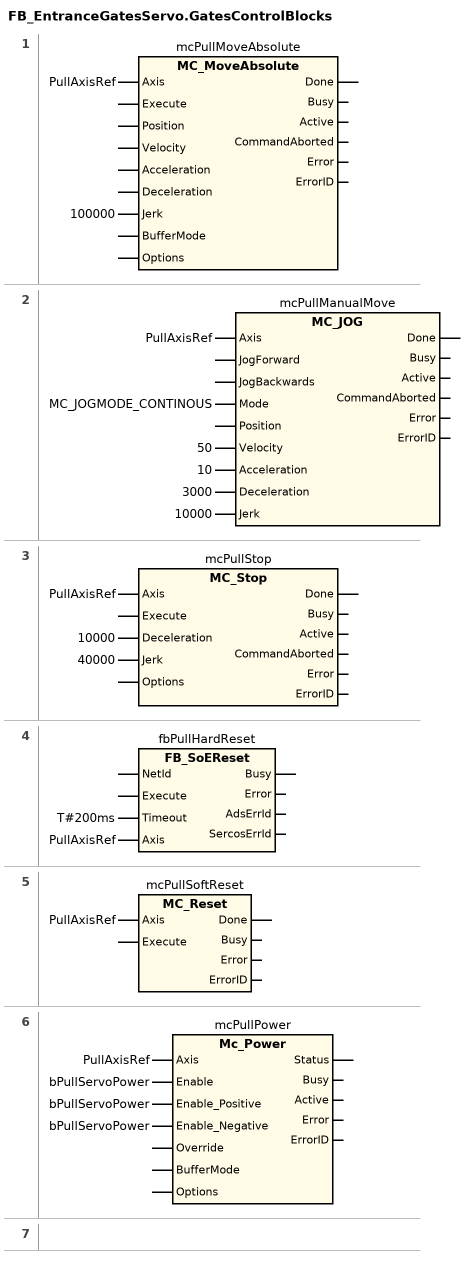
// NETWORK 1
mcPullMoveAbsolute(Axis := PullAxisRef, Jerk := 100000); // MC_MoveAbsolute

// NETWORK 2
mcPullManualMove(
    Axis := PullAxisRef,
    Mode := MC_JOGMODE_CONTINOUS,
    Velocity := 50,
    Acceleration := 10,
    Deceleration := 3000,
    Jerk := 10000); // MC_JOG

// NETWORK 3
mcPullStop(Axis := PullAxisRef, Deceleration := 10000, Jerk := 40000); // MC_Stop

// NETWORK 4
fbPullHardReset(Timeout := T#200ms, Axis := PullAxisRef); // FB_SoEReset

// NETWORK 5
mcPullSoftReset(Axis := PullAxisRef); // MC_Reset

// NETWORK 6
mcPullPower(
    Axis := PullAxisRef,
    Enable := bPullServoPower,
    Enable_Positive := bPullServoPower,
    Enable_Negative := bPullServoPower); // Mc_Power

// NETWORK 7
END_ACTION

ACTION Homing:
//Ustawienia początkowe
bGate1Actuator						:=	FALSE;
bGate2Actuator						:=	TRUE;

//Włączanie zasilania
mcPullPower.Override				:=	100;
mcPullManualMove.JogBackwards		:=	FALSE;
mcPullManualMove.JogForward			:=	FALSE;
bPullServoPower						:=	TRUE;

//Serwo włączone
IF mcPullPower.Status THEN
	
	//Ruch 
	mcPullMoveAbsolute.Velocity			:= lrPullVelocity;
	mcPullMoveAbsolute.Position			:= lrPullReadyPosition;
	mcPullMoveAbsolute.Acceleration		:= 1000;
	mcPullMoveAbsolute.Deceleration		:= 1000;
	mcPullMoveAbsolute.Execute			:= TRUE;

	//Wykonano ruch
	IF mcPullMoveAbsolute.Done THEN
		mcPullMoveAbsolute.Execute 		:=	FALSE;
		eState							:=	E_Station.eHomingDone;
	END_IF
END_IF
END_ACTION

ACTION ManualMovements:

//W trybie ruchów manualnych wykonuj ruchy za pomocą rozkazów manualnych
IF NOT bRun AND NOT bRunPrepare THEN
	bGate1Actuator					:=	bManualGate1Actuator;
	bGate2Actuator					:=	bManualGate2Actuator;	
	mcPullPower.Override			:=	100;
	mcPullManualMove.JogForward		:=	bManualPullRight;
	mcPullManualMove.JogBackwards	:=	bManualPullLeft;
ELSE	
	;
END_IF


IF bHoming OR bHeightSet THEN
	eState:=E_Station.eHoming;
END_IF
	

Running();


IF NOT bRun AND NOT bRunPrepare THEN
	bCycleDone 					:= FALSE;
	bCycleNotDone 				:= FALSE;			
	bCyclePrepareDone			:= FALSE;
END_IF
END_ACTION

ACTION Running:


CASE eRunningState OF
	
	//NIEGOTOWY
	E_EntranceGatesState.eDisabled:
			eRunningState:=E_EntranceGatesState.eReady;
		
	//ZGRZEWANIE GOTOWY DO PRACY
	E_EntranceGatesState.eReady:
		
		//Jeśli komenda podania platynki przejdź do stanu zasysania platynki
		IF NOT bCycleDone AND NOT bCycleNotDone THEN
			IF bBlocking THEN
				eRunningState := E_EntranceGatesState.eBlocking;	
			ELSIF bRun THEN
				eRunningState:=E_EntranceGatesState.ePulling;
			ELSIF bRunPrepare THEN
				eRunningState:=E_EntranceGatesState.ePullingToMiddle;				
			END_IF
		END_IF

	//Przesuwanie do środka (przyśpieszenie cyklu*)
	E_EntranceGatesState.ePullingToMiddle:
		
		bGate1Actuator:=TRUE;
		IF tonGate1Actuator.Q THEN //LU205
			bGate2Actuator:=FALSE;
		END_IF
		IF bOpenedGate1ActuatorSensor AND bClosedGate2ActuatorSensor THEN
			mcPullMoveAbsolute.Velocity			:=	lrPullVelocity;
			mcPullMoveAbsolute.Position			:=	lrPullStopOnePhasePosition/3;	
			mcPullMoveAbsolute.Acceleration		:=	lrPullAcceleration;
			mcPullMoveAbsolute.Deceleration		:=	lrPullDeceleration;
			IF rtPullingToMiddle.Q THEN
				mcPullMoveAbsolute.Execute		:=	TRUE;
			END_IF
			//Wykonano ruch
			IF mcPullMoveAbsolute.Done AND (lrPullActualPosition>mcPullMoveAbsolute.Position-6 AND lrPullActualPosition<mcPullMoveAbsolute.Position+6) THEN
				mcPullMoveAbsolute.Execute		:=	FALSE;
				eRunningState					:=	E_EntranceGatesState.ePullingToMiddleDone;			
			END_IF
		END_IF		

	//Koniec przesuwanie do środka (przyśpieszenie cyklu*)
	E_EntranceGatesState.ePullingToMiddleDone:	
		bCyclePrepareDone						:=	TRUE;
		IF bRun THEN
			eRunningState						:=	E_EntranceGatesState.ePulling; 
		END_IF
		
	//Rozpoczynanie przeciąganai
	E_EntranceGatesState.ePulling:
		
		bGate1Actuator:=TRUE;
		IF tonGate1Actuator.Q THEN //LU205
			bGate2Actuator:=FALSE;
		END_IF
		IF bOpenedGate1ActuatorSensor AND bClosedGate2ActuatorSensor THEN
		//Wpisanie przyśpieszeń przeciągania
			mcPullMoveAbsolute.Velocity			:=	lrPullVelocity;
			IF bMovingTwoForms AND bMovingThreeForms THEN 	(*przesuwanie do pozycji końcowej, trzy formatki*)
				mcPullMoveAbsolute.Position		:=	lrPullStopOnePhasePosition;
			ELSIF bMovingTwoForms THEN						(*przesuwanie do pozycji prawie końcowej, dwie formatki*)
				mcPullMoveAbsolute.Position		:=	(((lrPullStopOnePhasePosition-lrPullReadyPosition)*2/3)+lrPullReadyPosition);
			ELSE
				mcPullMoveAbsolute.Position		:=	lrPullStopTwoPhasePosition;
			END_IF	
			mcPullMoveAbsolute.Acceleration		:=	lrPullAcceleration;
			mcPullMoveAbsolute.Deceleration		:=	lrPullDeceleration;
			IF rtPulling.Q THEN
				mcPullMoveAbsolute.Execute		:=	TRUE;
			END_IF

			//Zamykanie szlabanu troche wcześniej
			IF  mcPullMoveAbsolute.Position - lrPullActualPosition < 100 THEN
				bGate2Actuator	:=	TRUE;
			END_IF
			
			//Wykonano ruch			
			IF mcPullMoveAbsolute.Done  AND lrPullActualPosition>mcPullMoveAbsolute.Position-3 AND lrPullActualPosition<mcPullMoveAbsolute.Position+3 THEN
				mcPullMoveAbsolute.Execute		:=	FALSE;
				eRunningState					:=	E_EntranceGatesState.ePullingDone;			
			END_IF
		END_IF
		
	//Koniec przeciągania
	E_EntranceGatesState.ePullingDone:
			bGate1Actuator	:=	FALSE;
			bGate2Actuator	:=	TRUE;
			IF bClosedGate1ActuatorSensor THEN
				bCycleDone		:=	TRUE;
				eRunningState:=E_EntranceGatesState.eReady; 
			END_IF

	//Blokowanie
	E_EntranceGatesState.eBlocking:
		bGate1Actuator:=FALSE;
		bGate2Actuator:=TRUE;
		IF (NOT bBlocking) OR (NOT bEnable) THEN 
			eRunningState:=E_EntranceGatesState.eReady;
		END_IF
		
END_CASE
END_ACTION

ACTION Statistics:



rtrigCycleTimerRead(CLK:=eRunningState=E_EntranceGatesState.eReady);
IF rtrigCycleTimerRead.Q THEN
	tCycleTime:=tonCycleTimer.ET;
END_IF
tonCycleTimer(IN:=eRunningState>E_EntranceGatesState.eReady,PT:=T#1D);
END_ACTION

END_FUNCTION_BLOCK

// ---- POUs/FB/FB_TankHeating.TcPOU
(*
Nazwa:			FB_TankHeating
Opis:			Stacja grzania zbiornika
Wersja:			v1.0
Data:			2019-07-02
Autor:			DP
Urzadzenia:		Podnosnik stacji, grzałka, silownik
Konfiguracja:	
Zmiany:
 - 20241214 [DP] Error = 0 
Info: 
- Dodano błędy od nastaw powyżej max i min (error 7 i 8)
- Dodano do testów inny regulator temperatury
- Zmiana Homingów według CatchStation
*)

FUNCTION_BLOCK FB_TankHeating
VAR_INPUT
	_CONTROL:BOOL;
	bEStop:BOOL;				//Stop Awaryjny nieaktywny
	bEnable:BOOL;				//Zezowlenie na pracę grzałki zasadniczej
	bRun:BOOL;
	bReset:BOOL;				//Reset błędu, jeśli w stanie "eError"
	bManualMode:BOOL; 			//Uruchomienie trybu ruchów ręcznych
	bIgnoreError:BOOL;			//Ignorowania błędów cyklu pracy

	_HEATER_PARAMETERS_:BOOL;	
	nHeaterTemperatureSV:INT;	//Zadana wartość grzałki grzałki zasadniczej
	rKp:REAL;					//Wzmocnienie proporcjonalne regulatora grzałki
	rTd:REAL;					//Czas różniczkowania regulatora grzałki
	rTi:REAL;					//Czas całkowania regulatora grzałki
	nTempHisteresis:INT;		//Dopuszczalna różnica pomiędzy wartością zadaną a aktualną [st. C]				
	
	_SENSORS_:BOOL;
	lrHeaterTemperatureCVSensor:LREAL;	//Wartość aktualna temperatury grzałki
	bTemperatureSensorFault:BOOL;		//Błąd czujnika temperatury

	iStationIndex:UDINT;				//Numer stacji 
	sStationName:WSTRING;				//Nazwa stacji
	
END_VAR
VAR_OUTPUT
	bHeaterPWMOut :BOOL;				//Wyjscie PWM sterujące grzałką
	eState: E_Station;					//Stan ogólny bloku
	eRunningState: E_MassHeatingState;	//Stan podbloku
	bError: BOOL;						//Błąd stacji
	nErrorNr: UDINT;					//Nr błędu grzałki zasadniczej
	sErrorDescription:STRING;			//Opis błędu
	sErrorStationName:STRING;			//Nazwa stacji
	bHomingDone:BOOL;					//Wymagane ponowne bazowanie (blad podczas bazowania lub stop awaryjny)
	tCycleTime:TIME;	
	bCycleDone:BOOL;
	bCycleNotDone:BOOL;
END_VAR
VAR
	fbTempRegulator: FB_TempRegulator;
	bTempRegulatorReset: BOOL;
	tonHeaterOnAndNotHeating: TON;
	lrHeaterTemperatureCVSensorLast:LREAL;	//Wartość aktualna temperatury grzałki
	tofbHeaterPWMOut: TOF;
	bStateError: BOOL;
	eLastState: E_Station;						//Stan ogólny bloku
	eLastRunningState: E_MassHeatingState;		//Stan podbloku
	eLastStateTemp: E_Station;					//Stan ogólny bloku
	eLastRunningStateTemp: E_MassHeatingState;	//Stan podbloku
	
	//Zmienne od EVENTLOGGER
	bAlarmInit 						: BOOL := TRUE; 
	nAlarmNumerator					: INT;
	arfbAlarm						: ARRAY[0..19] OF  FB_TcAlarm;		//Tablica bloczków błędów
	fbSourceInfo 					: FB_TcSourceInfo;
	iSourceInfo						: I_TcSourceInfo;
	sAlarmTest						: STRING;
	//Koniec zmiennych od EVENTLOGGER
	
END_VAR

VAR_IN_OUT

END_VAR

ErrorHandling();
Control();
HeaterRegulator();

(*Zapisywanie ostatniego stanu*)
IF eLastStateTemp<>eState THEN
	eLastState := eLastStateTemp;
END_IF
eLastStateTemp := eState;
IF eLastRunningStateTemp<>eRunningState THEN
	eLastRunningState := eLastRunningStateTemp;
END_IF
eLastRunningStateTemp := eRunningState;
(*Koniec Zapisywanie ostatniego stanu*)

ACTION Control:

	(*****Wyłączenie enable*****)
	IF NOT bEnable THEN
		IF eState <> E_Station.eDisabled AND eState <> E_Station.ePreparingToDisable THEN
				eState 				:= E_Station.ePreparingToDisable; 
		END_IF	
	END_IF

	(*****Estop*****)
	IF NOT bEstop  THEN	
		IF eState <> E_Station.eAborted AND eState <> E_Station.eAborting AND eState <> E_Station.eDisabled THEN
				eState 				:= E_Station.eAborting; 
		END_IF
	END_IF
	
	
	CASE eState OF
	/////////////////////////////	
		E_Station.eDisabled: 					// Stan nieaktywnosci (Stacja wyłączona) 
		
			IF bEnable THEN
				eState 				:= E_Station.ePreparingToReady; 
			END_IF 
			
    /////////////////////////////	    
		E_Station.eAborted: 					// Stan bezpiecznego zatrzymania (po Abortingu) 

			IF bEStop THEN
				eState 				:= E_Station.ePreparingToReady;
			END_IF
			
	/////////////////////////////	
		E_Station.eAborting:                 	// Stan bezpiecznego zatrzymywania (po EStopie)
		
			eState := E_Station.eAborted;  
			
	/////////////////////////////			
		E_Station.eError:                 	 	// Stan błędu 	
	
			IF bReset THEN
				eState 				:= E_Station.eResetting;
			END_IF
			
	/////////////////////////////
		E_Station.eResetting:					// Stan resetowania bledu (po Errorze)
			
			bError					:=	FALSE;
			IF NOT bError THEN
				nErrorNr 			:= 0;
   				sErrorDescription 	:= '';
				bTempRegulatorReset := FALSE;
				eState 				:= E_Station.ePreparingToReady;
			ELSE
				eState 				:= E_Station.eError;
			END_IF
        
	/////////////////////////////
		E_Station.eManualMovement:     			// Stan ruchów manualnych         
		
	/////////////////////////////
		E_Station.eHoming:						// Stan bazowania 
		
	/////////////////////////////
		E_Station.eHomingDone:                  // Stan wykonania bazowania 
		
	/////////////////////////////
		E_Station.ePreparingToReady:            // Stan przygotowywania do gotowosci (zawsze przed Ready)  
         
			eState:=E_Station.eReady;	
			
	/////////////////////////////
		E_Station.ePreparingToDisable:          // Stan przygotowywania do nieaktywnosci (po wyłączeniu Enable) 
                              
			eState 					:= E_Station.eDisabled; 
			
	/////////////////////////////
		E_Station.eReady:						// Stan gotowosci 
		
			IF bRun THEN
				eState 				:= E_Station.eStarting; 
			END_IF
			
	/////////////////////////////
		E_Station.eStopping:					// Stan zatrzymywania 
			
			Running();
			eState 					:= E_Station.eReady;	
			
	/////////////////////////////
		E_Station.eStarting:                  	// Stan uruchamiania (po Ready)
		
			eState					 := E_Station.eRunning; 
			
	/////////////////////////////
		E_Station.eRunning:               		// Stan wykonywania cyklu (po Startingu), w tym stanie osobny
 
			Running();
			IF NOT bRun THEN
				eState 				 := E_Station.eStopping;	
			END_IF
	/////////////////////////////		
	END_CASE
END_ACTION

